LIN {X 0,Y 473.765,Z 475.954,A -85,B 0,C 180,E1 -7294.679,E2 -7294.679} C_VEL
LIN {X 0,Y 473.866,Z 471.994,A -85,B 0,C 180,E1 -7295.958,E2 -7295.958} C_VEL
LIN {X 0,Y 474.033,Z 465.904,A -85,B 0,C 180,E1 -7297.452,E2 -7297.452} C_VEL
LIN {X 0,Y 474.322,Z 459.245,A -85,B 0,C 180,E1 -7298.734,E2 -7298.734} C_VEL
LIN {X 0,Y 474.676,Z 450.981,A -85,B 0,C 180,E1 -7300.017,E2 -7300.017} C_VEL
LIN {X 0,Y 475.049,Z 442.514,A -85,B 0,C 180,E1 -7301.087,E2 -7301.087} C_VEL
LIN {X 0,Y 475.614,Z 432.095,A -85,B 0,C 180,E1 -7302.15,E2 -7302.15} C_VEL
LIN {X 0,Y 476.019,Z 420.854,A -85,B 0,C 180,E1 -7303.075,E2 -7303.075} C_VEL
LIN {X 0,Y 476.498,Z 408.482,A -85,B 0,C 180,E1 -7303.866,E2 -7303.866} C_VEL
LIN {X 0,Y 476.994,Z 396.233,A -85,B 0,C 180,E1 -7304.45,E2 -7304.45} C_VEL
LIN {X 0,Y 477.32,Z 383.727,A -85,B 0,C 180,E1 -7304.876,E2 -7304.876} C_VEL
LIN {X 0,Y 477.558,Z 370.979,A -85,B 0,C 180,E1 -7305.141,E2 -7305.141} C_VEL
LIN {X 0,Y 478.059,Z 286.015,A -85,B 0,C 180,E1 -7306.443,E2 -7306.443} C_VEL
LIN {X 0,Y 475.428,Z 270.249,A -85,B 0,C 180,E1 -7306.808,E2 -7306.808} C_VEL
LIN {X 0,Y 475.47,Z 266.561,A -85,B 0,C 180,E1 -7307.415,E2 -7307.415} C_VEL
LIN {X 0,Y 476.068,Z 250.767,A -85,B 0,C 180,E1 -7310.298,E2 -7310.298} C_VEL
LIN {X 0,Y 476.598,Z 238.624,A -85,B 0,C 180,E1 -7312.543,E2 -7312.543} C_VEL
LIN {X 0,Y 474.683,Z 228.12,A -85,B 0,C 180,E1 -7314.665,E2 -7314.665} C_VEL
LIN {X 0,Y 474.645,Z 227.864,A -85,B 0,C 180,E1 -7315.428,E2 -7315.428} C_VEL
LIN {X 0,Y 474.644,Z 227.861,A -85,B 0,C 180,E1 -7318.281,E2 -7318.281} C_VEL
LIN {X 0,Y 474.6,Z 227.864,A -85,B 0,C 180,E1 -7321.216,E2 -7321.216} C_VEL
LIN {X 0,Y 474.633,Z 227.862,A -85,B 0,C 180,E1 -7324.239,E2 -7324.239} C_VEL
LIN {X 0,Y 474.585,Z 227.866,A -85,B 0,C 180,E1 -7327.382,E2 -7327.382} C_VEL
LIN {X 0,Y 474.615,Z 227.862,A -85,B 0,C 180,E1 -7330.656,E2 -7330.656} C_VEL
LIN {X 0,Y 474.591,Z 227.863,A -85,B 0,C 180,E1 -7333.477,E2 -7333.477} C_VEL
LIN {X 0,Y 474.591,Z 227.861,A -85,B 0,C 180,E1 -7336.518,E2 -7336.518} C_VEL
LIN {X 0,Y 474.593,Z 227.864,A -85,B 0,C 180,E1 -7339.337,E2 -7339.337} C_VEL
LIN {X 0,Y 474.604,Z 227.862,A -85,B 0,C 180,E1 -7341.702,E2 -7341.702} C_VEL
LIN {X 0,Y 474.619,Z 227.867,A -85,B 0,C 180,E1 -7344.723,E2 -7344.723} C_VEL
LIN {X 0,Y 474.631,Z 227.856,A -85,B 0,C 180,E1 -7347.785,E2 -7347.785} C_VEL
LIN {X 0,Y 474.602,Z 227.866,A -85,B 0,C 180,E1 -7350.886,E2 -7350.886} C_VEL
LIN {X 0,Y 474.586,Z 227.863,A -85,B 0,C 180,E1 -7353.621,E2 -7353.621} C_VEL
LIN {X 0,Y 474.628,Z 227.863,A -85,B 0,C 180,E1 -7356.639,E2 -7356.639} C_VEL
LIN {X 0,Y 474.643,Z 227.855,A -85,B 0,C 180,E1 -7360.086,E2 -7360.086} C_VEL
LIN {X 0,Y 474.623,Z 227.863,A -85,B 0,C 180,E1 -7362.771,E2 -7362.771} C_VEL
LIN {X 0,Y 474.623,Z 227.864,A -85,B 0,C 180,E1 -7365.417,E2 -7365.417} C_VEL
LIN {X 0,Y 474.694,Z 227.847,A -85,B 0,C 180,E1 -7368.034,E2 -7368.034} C_VEL
LIN {X 0,Y 474.682,Z 227.853,A -85,B 0,C 180,E1 -7371.483,E2 -7371.483} C_VEL
LIN {X 0,Y 474.743,Z 227.845,A -85,B 0,C 180,E1 -7374.049,E2 -7374.049} C_VEL
LIN {X 0,Y 474.855,Z 227.833,A -85,B 0,C 180,E1 -7377.452,E2 -7377.452} C_VEL
LIN {X 0,Y 474.86,Z 227.83,A -85,B 0,C 180,E1 -7379.997,E2 -7379.997} C_VEL
LIN {X 0,Y 474.856,Z 227.83,A -85,B 0,C 180,E1 -7382.541,E2 -7382.541} C_VEL
LIN {X 0,Y 474.717,Z 227.852,A -85,B 0,C 180,E1 -7385.945,E2 -7385.945} C_VEL
LIN {X 0,Y 474.688,Z 227.85,A -85,B 0,C 180,E1 -7388.511,E2 -7388.511} C_VEL
LIN {X 0,Y 474.683,Z 227.857,A -85,B 0,C 180,E1 -7391.959,E2 -7391.959} C_VEL
LIN {X 0,Y 474.657,Z 227.862,A -85,B 0,C 180,E1 -7395.764,E2 -7395.764} C_VEL
LIN {X 0,Y 474.637,Z 227.857,A -85,B 0,C 180,E1 -7399.007,E2 -7399.007} C_VEL
LIN {X 0,Y 474.562,Z 227.871,A -85,B 0,C 180,E1 -7401.726,E2 -7401.726} C_VEL
LIN {X 0,Y 474.611,Z 227.864,A -85,B 0,C 180,E1 -7404.491,E2 -7404.491} C_VEL
LIN {X 0,Y 474.652,Z 227.856,A -85,B 0,C 180,E1 -7407.331,E2 -7407.331} C_VEL
LIN {X 0,Y 474.573,Z 227.869,A -85,B 0,C 180,E1 -7410.807,E2 -7410.807} C_VEL
LIN {X 0,Y 474.606,Z 227.864,A -85,B 0,C 180,E1 -7413.981,E2 -7413.981} C_VEL
LIN {X 0,Y 474.543,Z 227.875,A -85,B 0,C 180,E1 -7416.897,E2 -7416.897} C_VEL
LIN {X 0,Y 474.62,Z 227.862,A -85,B 0,C 180,E1 -7419.649,E2 -7419.649} C_VEL
LIN {X 0,Y 474.615,Z 227.868,A -85,B 0,C 180,E1 -7422.928,E2 -7422.928} C_VEL
LIN {X 0,Y 474.605,Z 227.868,A -85,B 0,C 180,E1 -7426.243,E2 -7426.243} C_VEL
LIN {X 0,Y 474.634,Z 228.172,A -85,B 0,C 180,E1 -7426.508,E2 -7426.508} C_VEL
LIN {X 0,Y 476.004,Z 235.407,A -85,B 0,C 180,E1 -7428.002,E2 -7428.002} C_VEL
LIN {X 0,Y 475.688,Z 248.758,A -85,B 0,C 180,E1 -7430.56,E2 -7430.56} C_VEL
LIN {X 0,Y 475.414,Z 257.711,A -85,B 0,C 180,E1 -7432.212,E2 -7432.212} C_VEL
LIN {X 0,Y 476.311,Z 262.551,A -85,B 0,C 180,E1 -7432.363,E2 -7432.363} C_VEL
LIN {X 0,Y 478.228,Z 274.047,A -85,B 0,C 180,E1 -7432.616,E2 -7432.616} C_VEL
LIN {X 0,Y 477.488,Z 364.83,A -85,B 0,C 180,E1 -7434.019,E2 -7434.019} C_VEL
LIN {X 0,Y 477.188,Z 378.256,A -85,B 0,C 180,E1 -7434.396,E2 -7434.396} C_VEL
LIN {X 0,Y 476.867,Z 390.684,A -85,B 0,C 180,E1 -7434.918,E2 -7434.918} C_VEL
LIN {X 0,Y 476.416,Z 402.316,A -85,B 0,C 180,E1 -7435.575,E2 -7435.575} C_VEL
LIN {X 0,Y 476.347,Z 403.878,A -85,B 0,C 180,E1 -7435.681,E2 -7435.681} C_VEL
LIN {X 0,Y 475.493,Z 409.056,A -85,B 0,C 180,E1 -7436.025,E2 -7436.025} C_VEL
LIN {X 0,Y 472.367,Z 417.175,A -85,B 0,C 180,E1 -7436.603,E2 -7436.603} C_VEL
LIN {X 0,Y 469.192,Z 424.803,A -85,B 0,C 180,E1 -7437.257,E2 -7437.257} C_VEL
LIN {X 0,Y 468.251,Z 429.193,A -85,B 0,C 180,E1 -7437.72,E2 -7437.72} C_VEL
LIN {X 0,Y 467.764,Z 438.428,A -85,B 0,C 180,E1 -7438.905,E2 -7438.905} C_VEL
LIN {X 0,Y 467.323,Z 446.827,A -85,B 0,C 180,E1 -7440.248,E2 -7440.248} C_VEL
LIN {X 0,Y 467.12,Z 452.975,A -85,B 0,C 180,E1 -7441.467,E2 -7441.467} C_VEL
LIN {X 0,Y 466.95,Z 457.676,A -85,B 0,C 180,E1 -7442.611,E2 -7442.611} C_VEL
LIN {X 0,Y 466.765,Z 462.505,A -85,B 0,C 180,E1 -7444.112,E2 -7444.112} C_VEL
LIN {X 0,Y 466.632,Z 464.816,A -85,B 0,C 180,E1 -7445.059,E2 -7445.059} C_VEL
LIN {X 0,Y 466.503,Z 467.676,A -85,B 0,C 180,E1 -7446.764,E2 -7446.764} C_VEL
LIN {X 0,Y 466.46,Z 468.677,A -85,B 0,C 180,E1 -7447.874,E2 -7447.874} C_VEL
LIN {X 0,Y 466.492,Z 469.047,A -85,B 0,C 180,E1 -7449.063,E2 -7449.063} C_VEL
LIN {X 0,Y 466.512,Z 468.323,A -85,B 0,C 180,E1 -7450.646,E2 -7450.646} C_VEL
LIN {X 0,Y 466.551,Z 467.243,A -85,B 0,C 180,E1 -7451.608,E2 -7451.608} C_VEL
LIN {X 0,Y 466.584,Z 465.864,A -85,B 0,C 180,E1 -7452.469,E2 -7452.469} C_VEL
LIN {X 0,Y 466.737,Z 462.793,A -85,B 0,C 180,E1 -7453.827,E2 -7453.827} C_VEL
LIN {X 0,Y 466.861,Z 458.626,A -85,B 0,C 180,E1 -7455.174,E2 -7455.174} C_VEL
LIN {X 0,Y 467.074,Z 452.208,A -85,B 0,C 180,E1 -7456.736,E2 -7456.736} C_VEL
LIN {X 0,Y 467.434,Z 445.206,A -85,B 0,C 180,E1 -7458.07,E2 -7458.07} C_VEL
LIN {X 0,Y 467.697,Z 438.086,A -85,B 0,C 180,E1 -7459.175,E2 -7459.175} C_VEL
LIN {X 0,Y 468.144,Z 429.45,A -85,B 0,C 180,E1 -7460.278,E2 -7460.278} C_VEL
LIN {X 0,Y 468.644,Z 418.782,A -85,B 0,C 180,E1 -7461.377,E2 -7461.377} C_VEL
LIN {X 0,Y 469.181,Z 408.171,A -85,B 0,C 180,E1 -7462.254,E2 -7462.254} C_VEL
LIN {X 0,Y 469.622,Z 396.505,A -85,B 0,C 180,E1 -7463.017,E2 -7463.017} C_VEL
LIN {X 0,Y 470.048,Z 384.323,A -85,B 0,C 180,E1 -7463.617,E2 -7463.617} C_VEL
LIN {X 0,Y 470.405,Z 371.036,A -85,B 0,C 180,E1 -7464.079,E2 -7464.079} C_VEL
LIN {X 0,Y 470.584,Z 358.189,A -85,B 0,C 180,E1 -7464.35,E2 -7464.35} C_VEL
LIN {X 0,Y 471.037,Z 273.168,A -85,B 0,C 180,E1 -7465.669,E2 -7465.669} C_VEL
LIN {X 0,Y 468.41,Z 258.139,A -85,B 0,C 180,E1 -7466.022,E2 -7466.022} C_VEL
LIN {X 0,Y 468.814,Z 247.613,A -85,B 0,C 180,E1 -7468.068,E2 -7468.068} C_VEL
LIN {X 0,Y 469.142,Z 236.994,A -85,B 0,C 180,E1 -7470.216,E2 -7470.216} C_VEL
LIN {X 0,Y 467.744,Z 228.804,A -85,B 0,C 180,E1 -7472.019,E2 -7472.019} C_VEL
LIN {X 0,Y 467.593,Z 228.742,A -85,B 0,C 180,E1 -7473.448,E2 -7473.448} C_VEL
LIN {X 0,Y 467.696,Z 228.726,A -85,B 0,C 180,E1 -7476.039,E2 -7476.039} C_VEL
LIN {X 0,Y 467.639,Z 228.729,A -85,B 0,C 180,E1 -7478.645,E2 -7478.645} C_VEL
LIN {X 0,Y 467.641,Z 228.73,A -85,B 0,C 180,E1 -7482.147,E2 -7482.147} C_VEL
LIN {X 0,Y 467.609,Z 228.739,A -85,B 0,C 180,E1 -7485.887,E2 -7485.887} C_VEL
LIN {X 0,Y 467.584,Z 228.737,A -85,B 0,C 180,E1 -7489.311,E2 -7489.311} C_VEL
LIN {X 0,Y 467.496,Z 228.753,A -85,B 0,C 180,E1 -7492.077,E2 -7492.077} C_VEL
LIN {X 0,Y 467.533,Z 228.742,A -85,B 0,C 180,E1 -7494.893,E2 -7494.893} C_VEL
LIN {X 0,Y 467.544,Z 228.744,A -85,B 0,C 180,E1 -7497.775,E2 -7497.775} C_VEL
LIN {X 0,Y 467.534,Z 228.742,A -85,B 0,C 180,E1 -7501.048,E2 -7501.048} C_VEL
LIN {X 0,Y 467.544,Z 228.748,A -85,B 0,C 180,E1 -7504.243,E2 -7504.243} C_VEL
LIN {X 0,Y 467.492,Z 228.747,A -85,B 0,C 180,E1 -7507.186,E2 -7507.186} C_VEL
LIN {X 0,Y 467.529,Z 228.747,A -85,B 0,C 180,E1 -7510.271,E2 -7510.271} C_VEL
LIN {X 0,Y 467.521,Z 228.743,A -85,B 0,C 180,E1 -7513.75,E2 -7513.75} C_VEL
LIN {X 0,Y 467.524,Z 228.745,A -85,B 0,C 180,E1 -7516.259,E2 -7516.259} C_VEL
LIN {X 0,Y 467.538,Z 228.741,A -85,B 0,C 180,E1 -7519.738,E2 -7519.738} C_VEL
LIN {X 0,Y 467.529,Z 228.749,A -85,B 0,C 180,E1 -7522.818,E2 -7522.818} C_VEL
LIN {X 0,Y 467.561,Z 228.739,A -85,B 0,C 180,E1 -7525.764,E2 -7525.764} C_VEL
LIN {X 0,Y 467.535,Z 228.748,A -85,B 0,C 180,E1 -7528.964,E2 -7528.964} C_VEL
LIN {X 0,Y 467.534,Z 228.741,A -85,B 0,C 180,E1 -7532.23,E2 -7532.23} C_VEL
LIN {X 0,Y 467.545,Z 228.746,A -85,B 0,C 180,E1 -7535.114,E2 -7535.114} C_VEL
LIN {X 0,Y 467.525,Z 228.745,A -85,B 0,C 180,E1 -7537.93,E2 -7537.93} C_VEL
LIN {X 0,Y 467.615,Z 228.731,A -85,B 0,C 180,E1 -7540.696,E2 -7540.696} C_VEL
LIN {X 0,Y 467.636,Z 228.73,A -85,B 0,C 180,E1 -7544.309,E2 -7544.309} C_VEL
LIN {X 0,Y 467.647,Z 228.735,A -85,B 0,C 180,E1 -7547.858,E2 -7547.858} C_VEL
LIN {X 0,Y 467.638,Z 228.731,A -85,B 0,C 180,E1 -7551.36,E2 -7551.36} C_VEL
LIN {X 0,Y 467.703,Z 228.73,A -85,B 0,C 180,E1 -7553.966,E2 -7553.966} C_VEL
LIN {X 0,Y 467.817,Z 228.707,A -85,B 0,C 180,E1 -7557.42,E2 -7557.42} C_VEL
LIN {X 0,Y 467.854,Z 228.708,A -85,B 0,C 180,E1 -7560.003,E2 -7560.003} C_VEL
LIN {X 0,Y 467.817,Z 228.71,A -85,B 0,C 180,E1 -7562.586,E2 -7562.586} C_VEL
LIN {X 0,Y 467.71,Z 228.724,A -85,B 0,C 180,E1 -7566.041,E2 -7566.041} C_VEL
LIN {X 0,Y 467.644,Z 228.734,A -85,B 0,C 180,E1 -7568.646,E2 -7568.646} C_VEL
LIN {X 0,Y 467.667,Z 228.728,A -85,B 0,C 180,E1 -7572.148,E2 -7572.148} C_VEL
LIN {X 0,Y 467.661,Z 228.726,A -85,B 0,C 180,E1 -7575.887,E2 -7575.887} C_VEL
LIN {X 0,Y 467.633,Z 228.731,A -85,B 0,C 180,E1 -7579.31,E2 -7579.31} C_VEL
LIN {X 0,Y 467.544,Z 228.74,A -85,B 0,C 180,E1 -7582.076,E2 -7582.076} C_VEL
LIN {X 0,Y 467.57,Z 228.745,A -85,B 0,C 180,E1 -7584.892,E2 -7584.892} C_VEL
LIN {X 0,Y 467.56,Z 228.739,A -85,B 0,C 180,E1 -7587.775,E2 -7587.775} C_VEL
LIN {X 0,Y 467.561,Z 228.745,A -85,B 0,C 180,E1 -7591.042,E2 -7591.042} C_VEL
LIN {X 0,Y 467.59,Z 228.734,A -85,B 0,C 180,E1 -7594.241,E2 -7594.241} C_VEL
LIN {X 0,Y 467.556,Z 228.745,A -85,B 0,C 180,E1 -7597.186,E2 -7597.186} C_VEL
LIN {X 0,Y 467.572,Z 228.737,A -85,B 0,C 180,E1 -7600.268,E2 -7600.268} C_VEL
LIN {X 0,Y 467.559,Z 228.745,A -85,B 0,C 180,E1 -7603.746,E2 -7603.746} C_VEL
LIN {X 0,Y 467.558,Z 228.74,A -85,B 0,C 180,E1 -7606.255,E2 -7606.255} C_VEL
LIN {X 0,Y 467.571,Z 228.745,A -85,B 0,C 180,E1 -7609.733,E2 -7609.733} C_VEL
LIN {X 0,Y 467.556,Z 228.739,A -85,B 0,C 180,E1 -7612.815,E2 -7612.815} C_VEL
LIN {X 0,Y 467.598,Z 228.739,A -85,B 0,C 180,E1 -7616.212,E2 -7616.212} C_VEL
LIN {X 0,Y 467.58,Z 228.736,A -85,B 0,C 180,E1 -7619.266,E2 -7619.266} C_VEL
LIN {X 0,Y 467.617,Z 228.738,A -85,B 0,C 180,E1 -7622.468,E2 -7622.468} C_VEL
LIN {X 0,Y 467.639,Z 228.933,A -85,B 0,C 180,E1 -7625.202,E2 -7625.202} C_VEL
LIN {X 0,Y 469.538,Z 239.426,A -85,B 0,C 180,E1 -7627.329,E2 -7627.329} C_VEL
LIN {X 0,Y 469.006,Z 254.014,A -85,B 0,C 180,E1 -7630.067,E2 -7630.067} C_VEL
LIN {X 0,Y 468.383,Z 270.156,A -85,B 0,C 180,E1 -7633.013,E2 -7633.013} C_VEL
LIN {X 0,Y 471.181,Z 288.676,A -85,B 0,C 180,E1 -7633.429,E2 -7633.429} C_VEL
LIN {X 0,Y 470.481,Z 377.791,A -85,B 0,C 180,E1 -7634.817,E2 -7634.817} C_VEL
LIN {X 0,Y 470.119,Z 391.064,A -85,B 0,C 180,E1 -7635.193,E2 -7635.193} C_VEL
LIN {X 0,Y 469.669,Z 404.363,A -85,B 0,C 180,E1 -7635.76,E2 -7635.76} C_VEL
LIN {X 0,Y 469.2,Z 416.796,A -85,B 0,C 180,E1 -7636.497,E2 -7636.497} C_VEL
LIN {X 0,Y 468.768,Z 427.881,A -85,B 0,C 180,E1 -7637.341,E2 -7637.341} C_VEL
LIN {X 0,Y 468.257,Z 438.115,A -85,B 0,C 180,E1 -7638.309,E2 -7638.309} C_VEL
LIN {X 0,Y 467.772,Z 447.372,A -85,B 0,C 180,E1 -7639.393,E2 -7639.393} C_VEL
LIN {X 0,Y 467.341,Z 456.36,A -85,B 0,C 180,E1 -7640.695,E2 -7640.695} C_VEL
LIN {X 0,Y 467.057,Z 463.597,A -85,B 0,C 180,E1 -7641.998,E2 -7641.998} C_VEL
LIN {X 0,Y 466.862,Z 468.48,A -85,B 0,C 180,E1 -7643.082,E2 -7643.082} C_VEL
LIN {X 0,Y 466.793,Z 473.226,A -85,B 0,C 180,E1 -7644.383,E2 -7644.383} C_VEL
LIN {X 0,Y 466.65,Z 476.851,A -85,B 0,C 180,E1 -7645.68,E2 -7645.68} C_VEL
LIN {X 0,Y 466.663,Z 478.725,A -85,B 0,C 180,E1 -7646.545,E2 -7646.545} C_VEL
LIN {X 0,Y 466.647,Z 480.132,A -85,B 0,C 180,E1 -7647.409,E2 -7647.409} C_VEL
LIN {X 0,Y 466.592,Z 481.747,A -85,B 0,C 180,E1 -7649.136,E2 -7649.136} C_VEL
LIN {X 0,Y 466.601,Z 481.972,A -85,B 0,C 180,E1 -7649.999,E2 -7649.999} C_VEL
LIN {X 0,Y 466.592,Z 481.766,A -85,B 0,C 180,E1 -7650.862,E2 -7650.862} C_VEL
LIN {X 0,Y 466.646,Z 480.176,A -85,B 0,C 180,E1 -7652.588,E2 -7652.588} C_VEL
LIN {X 0,Y 466.663,Z 478.789,A -85,B 0,C 180,E1 -7653.452,E2 -7653.452} C_VEL
LIN {X 0,Y 466.693,Z 475.866,A -85,B 0,C 180,E1 -7654.75,E2 -7654.75} C_VEL
LIN {X 0,Y 466.78,Z 471.908,A -85,B 0,C 180,E1 -7656.048,E2 -7656.048} C_VEL
LIN {X 0,Y 466.983,Z 465.823,A -85,B 0,C 180,E1 -7657.566,E2 -7657.566} C_VEL
LIN {X 0,Y 467.288,Z 459.175,A -85,B 0,C 180,E1 -7658.867,E2 -7658.867} C_VEL
LIN {X 0,Y 467.636,Z 450.933,A -85,B 0,C 180,E1 -7660.17,E2 -7660.17} C_VEL
LIN {X 0,Y 468.084,Z 442.497,A -85,B 0,C 180,E1 -7661.254,E2 -7661.254} C_VEL
LIN {X 0,Y 468.658,Z 432.316,A -85,B 0,C 180,E1 -7662.315,E2 -7662.315} C_VEL
LIN {X 0,Y 469.022,Z 422.073,A -85,B 0,C 180,E1 -7663.186,E2 -7663.186} C_VEL
LIN {X 0,Y 469.529,Z 410.519,A -85,B 0,C 180,E1 -7663.965,E2 -7663.965} C_VEL
LIN {X 0,Y 470.047,Z 399.055,A -85,B 0,C 180,E1 -7664.557,E2 -7664.557} C_VEL
LIN {X 0,Y 470.387,Z 385.936,A -85,B 0,C 180,E1 -7665.045,E2 -7665.045} C_VEL
LIN {X 0,Y 470.747,Z 373.321,A -85,B 0,C 180,E1 -7665.338,E2 -7665.338} C_VEL
LIN {X 0,Y 471.274,Z 286.938,A -85,B 0,C 180,E1 -7666.686,E2 -7666.686} C_VEL
LIN {X 0,Y 468.441,Z 269.969,A -85,B 0,C 180,E1 -7667.094,E2 -7667.094} C_VEL
LIN {X 0,Y 469.038,Z 254.391,A -85,B 0,C 180,E1 -7669.929,E2 -7669.929} C_VEL
LIN {X 0,Y 469.657,Z 239.86,A -85,B 0,C 180,E1 -7672.662,E2 -7672.662} C_VEL
LIN {X 0,Y 467.677,Z 229.048,A -85,B 0,C 180,E1 -7674.881,E2 -7674.881} C_VEL
LIN {X 0,Y 467.616,Z 228.739,A -85,B 0,C 180,E1 -7675.306,E2 -7675.306} C_VEL
LIN {X 0,Y 467.619,Z 228.739,A -85,B 0,C 180,E1 -7677.767,E2 -7677.767} C_VEL
LIN {X 0,Y 467.569,Z 228.739,A -85,B 0,C 180,E1 -7681.042,E2 -7681.042} C_VEL
LIN {X 0,Y 467.59,Z 228.739,A -85,B 0,C 180,E1 -7684.24,E2 -7684.24} C_VEL
LIN {X 0,Y 467.543,Z 228.743,A -85,B 0,C 180,E1 -7687.183,E2 -7687.183} C_VEL
LIN {X 0,Y 467.57,Z 228.744,A -85,B 0,C 180,E1 -7690.263,E2 -7690.263} C_VEL
LIN {X 0,Y 467.561,Z 228.741,A -85,B 0,C 180,E1 -7692.561,E2 -7692.561} C_VEL
LIN {X 0,Y 467.565,Z 228.738,A -85,B 0,C 180,E1 -7695.05,E2 -7695.05} C_VEL
LIN {X 0,Y 467.565,Z 228.745,A -85,B 0,C 180,E1 -7698.593,E2 -7698.593} C_VEL
LIN {X 0,Y 467.559,Z 228.741,A -85,B 0,C 180,E1 -7701.952,E2 -7701.952} C_VEL
LIN {X 0,Y 467.559,Z 228.741,A -85,B 0,C 180,E1 -7705.164,E2 -7705.164} C_VEL
LIN {X 0,Y 467.578,Z 228.738,A -85,B 0,C 180,E1 -7708.257,E2 -7708.257} C_VEL
LIN {X 0,Y 467.549,Z 228.742,A -85,B 0,C 180,E1 -7711.246,E2 -7711.246} C_VEL
LIN {X 0,Y 467.562,Z 228.739,A -85,B 0,C 180,E1 -7714.155,E2 -7714.155} C_VEL
LIN {X 0,Y 467.565,Z 228.745,A -85,B 0,C 180,E1 -7716.993,E2 -7716.993} C_VEL
LIN {X 0,Y 467.613,Z 228.731,A -85,B 0,C 180,E1 -7719.774,E2 -7719.774} C_VEL
LIN {X 0,Y 467.585,Z 228.737,A -85,B 0,C 180,E1 -7722.503,E2 -7722.503} C_VEL
LIN {X 0,Y 467.585,Z 228.744,A -85,B 0,C 180,E1 -7725.193,E2 -7725.193} C_VEL
LIN {X 0,Y 467.646,Z 228.726,A -85,B 0,C 180,E1 -7727.851,E2 -7727.851} C_VEL
LIN {X 0,Y 467.642,Z 228.732,A -85,B 0,C 180,E1 -7731.353,E2 -7731.353} C_VEL
LIN {X 0,Y 467.708,Z 228.722,A -85,B 0,C 180,E1 -7733.959,E2 -7733.959} C_VEL
LIN {X 0,Y 467.795,Z 228.712,A -85,B 0,C 180,E1 -7737.414,E2 -7737.414} C_VEL
LIN {X 0,Y 467.83,Z 228.706,A -85,B 0,C 180,E1 -7739.997,E2 -7739.997} C_VEL
LIN {X 0,Y 467.797,Z 228.709,A -85,B 0,C 180,E1 -7742.58,E2 -7742.58} C_VEL
LIN {X 0,Y 467.682,Z 228.727,A -85,B 0,C 180,E1 -7746.035,E2 -7746.035} C_VEL
LIN {X 0,Y 467.647,Z 228.727,A -85,B 0,C 180,E1 -7748.64,E2 -7748.64} C_VEL
LIN {X 0,Y 467.635,Z 228.732,A -85,B 0,C 180,E1 -7752.142,E2 -7752.142} C_VEL
LIN {X 0,Y 467.626,Z 228.737,A -85,B 0,C 180,E1 -7755.881,E2 -7755.881} C_VEL
LIN {X 0,Y 467.596,Z 228.735,A -85,B 0,C 180,E1 -7759.305,E2 -7759.305} C_VEL
LIN {X 0,Y 467.508,Z 228.752,A -85,B 0,C 180,E1 -7762.071,E2 -7762.071} C_VEL
LIN {X 0,Y 467.556,Z 228.739,A -85,B 0,C 180,E1 -7764.885,E2 -7764.885} C_VEL
LIN {X 0,Y 467.591,Z 228.737,A -85,B 0,C 180,E1 -7767.766,E2 -7767.766} C_VEL
LIN {X 0,Y 467.537,Z 228.744,A -85,B 0,C 180,E1 -7771.042,E2 -7771.042} C_VEL
LIN {X 0,Y 467.558,Z 228.745,A -85,B 0,C 180,E1 -7774.24,E2 -7774.24} C_VEL
LIN {X 0,Y 467.518,Z 228.747,A -85,B 0,C 180,E1 -7777.184,E2 -7777.184} C_VEL
LIN {X 0,Y 467.562,Z 228.744,A -85,B 0,C 180,E1 -7780.26,E2 -7780.26} C_VEL
LIN {X 0,Y 467.583,Z 228.742,A -85,B 0,C 180,E1 -7782.569,E2 -7782.569} C_VEL
LIN {X 0,Y 467.589,Z 228.823,A -85,B 0,C 180,E1 -7786.214,E2 -7786.214} C_VEL
LIN {X 0,Y 469.088,Z 236.967,A -85,B 0,C 180,E1 -7787.953,E2 -7787.953} C_VEL
LIN {X 0,Y 468.743,Z 249.657,A -85,B 0,C 180,E1 -7790.418,E2 -7790.418} C_VEL
LIN {X 0,Y 468.48,Z 257.715,A -85,B 0,C 180,E1 -7791.928,E2 -7791.928} C_VEL
LIN {X 0,Y 468.99,Z 260.702,A -85,B 0,C 180,E1 -7792.045,E2 -7792.045} C_VEL
LIN {X 0,Y 471.426,Z 273.939,A -85,B 0,C 180,E1 -7792.353,E2 -7792.353} C_VEL
LIN {X 0,Y 470.659,Z 365.908,A -85,B 0,C 180,E1 -7793.804,E2 -7793.804} C_VEL
LIN {X 0,Y 470.329,Z 379.436,A -85,B 0,C 180,E1 -7794.202,E2 -7794.202} C_VEL
LIN {X 0,Y 470.01,Z 391.404,A -85,B 0,C 180,E1 -7794.723,E2 -7794.723} C_VEL
LIN {X 0,Y 469.507,Z 403.103,A -85,B 0,C 180,E1 -7795.406,E2 -7795.406} C_VEL
LIN {X 0,Y 468.978,Z 413.717,A -85,B 0,C 180,E1 -7796.198,E2 -7796.198} C_VEL
LIN {X 0,Y 468.514,Z 423.803,A -85,B 0,C 180,E1 -7797.134,E2 -7797.134} C_VEL
LIN {X 0,Y 468.251,Z 429.193,A -85,B 0,C 180,E1 -7797.72,E2 -7797.72} C_VEL
LIN {X 0,Y 467.306,Z 433.457,A -85,B 0,C 180,E1 -7798.21,E2 -7798.21} C_VEL
LIN {X 0,Y 464.097,Z 440.035,A -85,B 0,C 180,E1 -7799.037,E2 -7799.037} C_VEL
LIN {X 0,Y 461.001,Z 445.992,A -85,B 0,C 180,E1 -7799.94,E2 -7799.94} C_VEL
LIN {X 0,Y 460.238,Z 449.28,A -85,B 0,C 180,E1 -7800.542,E2 -7800.542} C_VEL
LIN {X 0,Y 460.004,Z 454.792,A -85,B 0,C 180,E1 -7801.732,E2 -7801.732} C_VEL
LIN {X 0,Y 459.78,Z 460.175,A -85,B 0,C 180,E1 -7803.199,E2 -7803.199} C_VEL
LIN {X 0,Y 459.599,Z 464.172,A -85,B 0,C 180,E1 -7804.651,E2 -7804.651} C_VEL
LIN {X 0,Y 459.486,Z 466.143,A -85,B 0,C 180,E1 -7805.61,E2 -7805.61} C_VEL
LIN {X 0,Y 459.428,Z 467.622,A -85,B 0,C 180,E1 -7806.598,E2 -7806.598} C_VEL
LIN {X 0,Y 459.37,Z 468.565,A -85,B 0,C 180,E1 -7807.514,E2 -7807.514} C_VEL
LIN {X 0,Y 459.404,Z 469.136,A -85,B 0,C 180,E1 -7808.921,E2 -7808.921} C_VEL
LIN {X 0,Y 459.43,Z 468.684,A -85,B 0,C 180,E1 -7810.336,E2 -7810.336} C_VEL
LIN {X 0,Y 459.45,Z 467.524,A -85,B 0,C 180,E1 -7811.494,E2 -7811.494} C_VEL
LIN {X 0,Y 459.541,Z 464.751,A -85,B 0,C 180,E1 -7813.109,E2 -7813.109} C_VEL
LIN {X 0,Y 459.696,Z 461.507,A -85,B 0,C 180,E1 -7814.38,E2 -7814.38} C_VEL
LIN {X 0,Y 459.849,Z 456.545,A -85,B 0,C 180,E1 -7815.847,E2 -7815.847} C_VEL
LIN {X 0,Y 460.167,Z 449.428,A -85,B 0,C 180,E1 -7817.431,E2 -7817.431} C_VEL
LIN {X 0,Y 460.513,Z 441.734,A -85,B 0,C 180,E1 -7818.781,E2 -7818.781} C_VEL
LIN {X 0,Y 460.934,Z 433.851,A -85,B 0,C 180,E1 -7819.903,E2 -7819.903} C_VEL
LIN {X 0,Y 461.399,Z 424.226,A -85,B 0,C 180,E1 -7821.019,E2 -7821.019} C_VEL
LIN {X 0,Y 461.953,Z 413.581,A -85,B 0,C 180,E1 -7822.016,E2 -7822.016} C_VEL
LIN {X 0,Y 462.457,Z 403.178,A -85,B 0,C 180,E1 -7822.799,E2 -7822.799} C_VEL
LIN {X 0,Y 462.968,Z 390.897,A -85,B 0,C 180,E1 -7823.519,E2 -7823.519} C_VEL
LIN {X 0,Y 463.308,Z 378.046,A -85,B 0,C 180,E1 -7824.07,E2 -7824.07} C_VEL
LIN {X 0,Y 463.638,Z 365.538,A -85,B 0,C 180,E1 -7824.429,E2 -7824.429} C_VEL
LIN {X 0,Y 464.212,Z 273.918,A -85,B 0,C 180,E1 -7825.891,E2 -7825.891} C_VEL
LIN {X 0,Y 461.43,Z 258.269,A -85,B 0,C 180,E1 -7826.263,E2 -7826.263} C_VEL
LIN {X 0,Y 461.672,Z 252.419,A -85,B 0,C 180,E1 -7827.384,E2 -7827.384} C_VEL
LIN {X 0,Y 462.213,Z 239.599,A -85,B 0,C 180,E1 -7830.001,E2 -7830.001} C_VEL
LIN {X 0,Y 461.573,Z 234.503,A -85,B 0,C 180,E1 -7831.092,E2 -7831.092} C_VEL
LIN {X 0,Y 460.711,Z 229.692,A -85,B 0,C 180,E1 -7832.187,E2 -7832.187} C_VEL
LIN {X 0,Y 460.654,Z 229.607,A -85,B 0,C 180,E1 -7835.253,E2 -7835.253} C_VEL
LIN {X 0,Y 460.653,Z 229.602,A -85,B 0,C 180,E1 -7837.893,E2 -7837.893} C_VEL
LIN {X 0,Y 460.587,Z 229.613,A -85,B 0,C 180,E1 -7841.443,E2 -7841.443} C_VEL
LIN {X 0,Y 460.511,Z 229.619,A -85,B 0,C 180,E1 -7844.135,E2 -7844.135} C_VEL
LIN {X 0,Y 460.524,Z 229.615,A -85,B 0,C 180,E1 -7846.857,E2 -7846.857} C_VEL
LIN {X 0,Y 460.53,Z 229.619,A -85,B 0,C 180,E1 -7849.618,E2 -7849.618} C_VEL
LIN {X 0,Y 460.473,Z 229.624,A -85,B 0,C 180,E1 -7852.432,E2 -7852.432} C_VEL
LIN {X 0,Y 460.51,Z 229.621,A -85,B 0,C 180,E1 -7855.799,E2 -7855.799} C_VEL
LIN {X 0,Y 460.491,Z 229.626,A -85,B 0,C 180,E1 -7858.238,E2 -7858.238} C_VEL
LIN {X 0,Y 460.488,Z 229.619,A -85,B 0,C 180,E1 -7861.286,E2 -7861.286} C_VEL
LIN {X 0,Y 460.489,Z 229.626,A -85,B 0,C 180,E1 -7864.507,E2 -7864.507} C_VEL
LIN {X 0,Y 460.456,Z 229.623,A -85,B 0,C 180,E1 -7867.629,E2 -7867.629} C_VEL
LIN {X 0,Y 460.489,Z 229.622,A -85,B 0,C 180,E1 -7871.017,E2 -7871.017} C_VEL
LIN {X 0,Y 460.487,Z 229.627,A -85,B 0,C 180,E1 -7874.594,E2 -7874.594} C_VEL
LIN {X 0,Y 460.47,Z 229.621,A -85,B 0,C 180,E1 -7877.819,E2 -7877.819} C_VEL
LIN {X 0,Y 460.493,Z 229.619,A -85,B 0,C 180,E1 -7880.14,E2 -7880.14} C_VEL
LIN {X 0,Y 460.459,Z 229.625,A -85,B 0,C 180,E1 -7883.475,E2 -7883.475} C_VEL
LIN {X 0,Y 460.501,Z 229.621,A -85,B 0,C 180,E1 -7886.678,E2 -7886.678} C_VEL
LIN {X 0,Y 460.49,Z 229.62,A -85,B 0,C 180,E1 -7889.764,E2 -7889.764} C_VEL
LIN {X 0,Y 460.478,Z 229.623,A -85,B 0,C 180,E1 -7892.755,E2 -7892.755} C_VEL
LIN {X 0,Y 460.507,Z 229.621,A -85,B 0,C 180,E1 -7895.671,E2 -7895.671} C_VEL
LIN {X 0,Y 460.516,Z 229.616,A -85,B 0,C 180,E1 -7898.583,E2 -7898.583} C_VEL
LIN {X 0,Y 460.579,Z 229.613,A -85,B 0,C 180,E1 -7901.315,E2 -7901.315} C_VEL
LIN {X 0,Y 460.584,Z 229.61,A -85,B 0,C 180,E1 -7904.062,E2 -7904.062} C_VEL
LIN {X 0,Y 460.603,Z 229.613,A -85,B 0,C 180,E1 -7907.67,E2 -7907.67} C_VEL
LIN {X 0,Y 460.593,Z 229.607,A -85,B 0,C 180,E1 -7911.227,E2 -7911.227} C_VEL
LIN {X 0,Y 460.67,Z 229.604,A -85,B 0,C 180,E1 -7913.873,E2 -7913.873} C_VEL
LIN {X 0,Y 460.761,Z 229.586,A -85,B 0,C 180,E1 -7917.381,E2 -7917.381} C_VEL
LIN {X 0,Y 460.824,Z 229.584,A -85,B 0,C 180,E1 -7920.003,E2 -7920.003} C_VEL
LIN {X 0,Y 460.761,Z 229.589,A -85,B 0,C 180,E1 -7922.626,E2 -7922.626} C_VEL
LIN {X 0,Y 460.676,Z 229.601,A -85,B 0,C 180,E1 -7926.134,E2 -7926.134} C_VEL
LIN {X 0,Y 460.599,Z 229.609,A -85,B 0,C 180,E1 -7928.78,E2 -7928.78} C_VEL
LIN {X 0,Y 460.621,Z 229.608,A -85,B 0,C 180,E1 -7932.337,E2 -7932.337} C_VEL
LIN {X 0,Y 460.614,Z 229.604,A -85,B 0,C 180,E1 -7936,E2 -7936} C_VEL
LIN {X 0,Y 460.579,Z 229.608,A -85,B 0,C 180,E1 -7939.618,E2 -7939.618} C_VEL
LIN {X 0,Y 460.521,Z 229.618,A -85,B 0,C 180,E1 -7942.431,E2 -7942.431} C_VEL
LIN {X 0,Y 460.547,Z 229.612,A -85,B 0,C 180,E1 -7945.794,E2 -7945.794} C_VEL
LIN {X 0,Y 460.534,Z 229.621,A -85,B 0,C 180,E1 -7949.234,E2 -7949.234} C_VEL
LIN {X 0,Y 460.532,Z 229.614,A -85,B 0,C 180,E1 -7952.287,E2 -7952.287} C_VEL
LIN {X 0,Y 460.519,Z 229.622,A -85,B 0,C 180,E1 -7955.447,E2 -7955.447} C_VEL
LIN {X 0,Y 460.518,Z 229.617,A -85,B 0,C 180,E1 -7958.892,E2 -7958.892} C_VEL
LIN {X 0,Y 460.517,Z 229.623,A -85,B 0,C 180,E1 -7961.599,E2 -7961.599} C_VEL
LIN {X 0,Y 460.525,Z 229.614,A -85,B 0,C 180,E1 -7964.59,E2 -7964.59} C_VEL
LIN {X 0,Y 460.489,Z 229.627,A -85,B 0,C 180,E1 -7967.813,E2 -7967.813} C_VEL
LIN {X 0,Y 460.526,Z 229.618,A -85,B 0,C 180,E1 -7970.136,E2 -7970.136} C_VEL
LIN {X 0,Y 460.486,Z 229.622,A -85,B 0,C 180,E1 -7973.47,E2 -7973.47} C_VEL
LIN {X 0,Y 460.542,Z 229.613,A -85,B 0,C 180,E1 -7976.675,E2 -7976.675} C_VEL
LIN {X 0,Y 460.52,Z 229.619,A -85,B 0,C 180,E1 -7979.759,E2 -7979.759} C_VEL
LIN {X 0,Y 460.547,Z 229.619,A -85,B 0,C 180,E1 -7982.753,E2 -7982.753} C_VEL
LIN {X 0,Y 460.594,Z 229.796,A -85,B 0,C 180,E1 -7985.008,E2 -7985.008} C_VEL
LIN {X 0,Y 462.556,Z 240.445,A -85,B 0,C 180,E1 -7987.203,E2 -7987.203} C_VEL
LIN {X 0,Y 462.146,Z 251.389,A -85,B 0,C 180,E1 -7989.293,E2 -7989.293} C_VEL
LIN {X 0,Y 461.521,Z 265.951,A -85,B 0,C 180,E1 -7992.038,E2 -7992.038} C_VEL
LIN {X 0,Y 461.396,Z 270.235,A -85,B 0,C 180,E1 -7992.776,E2 -7992.776} C_VEL
LIN {X 0,Y 464.359,Z 288.708,A -85,B 0,C 180,E1 -7993.191,E2 -7993.191} C_VEL
LIN {X 0,Y 463.583,Z 378.085,A -85,B 0,C 180,E1 -7994.614,E2 -7994.614} C_VEL
LIN {X 0,Y 463.187,Z 391.99,A -85,B 0,C 180,E1 -7995.023,E2 -7995.023} C_VEL
LIN {X 0,Y 462.73,Z 404.96,A -85,B 0,C 180,E1 -7995.598,E2 -7995.598} C_VEL
LIN {X 0,Y 462.226,Z 417.548,A -85,B 0,C 180,E1 -7996.367,E2 -7996.367} C_VEL
LIN {X 0,Y 461.782,Z 428.246,A -85,B 0,C 180,E1 -7997.204,E2 -7997.204} C_VEL
LIN {X 0,Y 461.26,Z 437.844,A -85,B 0,C 180,E1 -7998.129,E2 -7998.129} C_VEL
LIN {X 0,Y 460.773,Z 447.148,A -85,B 0,C 180,E1 -7999.23,E2 -7999.23} C_VEL
LIN {X 0,Y 460.297,Z 456.169,A -85,B 0,C 180,E1 -8000.552,E2 -8000.552} C_VEL
LIN {X 0,Y 460.013,Z 463.433,A -85,B 0,C 180,E1 -8001.874,E2 -8001.874} C_VEL
LIN {X 0,Y 459.782,Z 468.333,A -85,B 0,C 180,E1 -8002.975,E2 -8002.975} C_VEL
LIN {X 0,Y 459.691,Z 473.094,A -85,B 0,C 180,E1 -8004.295,E2 -8004.295} C_VEL
LIN {X 0,Y 459.568,Z 476.731,A -85,B 0,C 180,E1 -8005.613,E2 -8005.613} C_VEL
LIN {X 0,Y 459.56,Z 478.61,A -85,B 0,C 180,E1 -8006.492,E2 -8006.492} C_VEL
LIN {X 0,Y 459.569,Z 480.024,A -85,B 0,C 180,E1 -8007.369,E2 -8007.369} C_VEL
LIN {X 0,Y 459.497,Z 481.644,A -85,B 0,C 180,E1 -8009.122,E2 -8009.122} C_VEL
LIN {X 0,Y 459.504,Z 481.873,A -85,B 0,C 180,E1 -8009.999,E2 -8009.999} C_VEL
LIN {X 0,Y 459.497,Z 481.671,A -85,B 0,C 180,E1 -8010.875,E2 -8010.875} C_VEL
LIN {X 0,Y 459.569,Z 480.088,A -85,B 0,C 180,E1 -8012.628,E2 -8012.628} C_VEL
LIN {X 0,Y 459.56,Z 478.706,A -85,B 0,C 180,E1 -8013.506,E2 -8013.506} C_VEL
LIN {X 0,Y 459.625,Z 475.792,A -85,B 0,C 180,E1 -8014.823,E2 -8014.823} C_VEL
LIN {X 0,Y 459.704,Z 471.848,A -85,B 0,C 180,E1 -8016.142,E2 -8016.142} C_VEL
LIN {X 0,Y 459.871,Z 466.774,A -85,B 0,C 180,E1 -8017.462,E2 -8017.462} C_VEL
LIN {X 0,Y 460.175,Z 460.392,A -85,B 0,C 180,E1 -8018.783,E2 -8018.783} C_VEL
LIN {X 0,Y 460.572,Z 452.42,A -85,B 0,C 180,E1 -8020.105,E2 -8020.105} C_VEL
LIN {X 0,Y 460.97,Z 444.305,A -85,B 0,C 180,E1 -8021.207,E2 -8021.207} C_VEL
LIN {X 0,Y 461.558,Z 434.413,A -85,B 0,C 180,E1 -8022.307,E2 -8022.307} C_VEL
LIN {X 0,Y 462.063,Z 423.443,A -85,B 0,C 180,E1 -8023.287,E2 -8023.287} C_VEL
LIN {X 0,Y 462.583,Z 412.416,A -85,B 0,C 180,E1 -8024.067,E2 -8024.067} C_VEL
LIN {X 0,Y 463.156,Z 400.404,A -85,B 0,C 180,E1 -8024.723,E2 -8024.723} C_VEL
LIN {X 0,Y 463.509,Z 388.122,A -85,B 0,C 180,E1 -8025.217,E2 -8025.217} C_VEL
LIN {X 0,Y 463.907,Z 375.514,A -85,B 0,C 180,E1 -8025.541,E2 -8025.541} C_VEL
LIN {X 0,Y 464.481,Z 287.566,A -85,B 0,C 180,E1 -8026.943,E2 -8026.943} C_VEL
LIN {X 0,Y 461.496,Z 269.83,A -85,B 0,C 180,E1 -8027.38,E2 -8027.38} C_VEL
LIN {X 0,Y 462.131,Z 254.416,A -85,B 0,C 180,E1 -8030.24,E2 -8030.24} C_VEL
LIN {X 0,Y 462.747,Z 242.307,A -85,B 0,C 180,E1 -8032.548,E2 -8032.548} C_VEL
LIN {X 0,Y 461.654,Z 235.11,A -85,B 0,C 180,E1 -8034.016,E2 -8034.016} C_VEL
LIN {X 0,Y 460.6,Z 229.778,A -85,B 0,C 180,E1 -8035.17,E2 -8035.17} C_VEL
LIN {X 0,Y 460.552,Z 229.617,A -85,B 0,C 180,E1 -8038.231,E2 -8038.231} C_VEL
LIN {X 0,Y 460.523,Z 229.619,A -85,B 0,C 180,E1 -8041.28,E2 -8041.28} C_VEL
LIN {X 0,Y 460.533,Z 229.615,A -85,B 0,C 180,E1 -8044.503,E2 -8044.503} C_VEL
LIN {X 0,Y 460.499,Z 229.623,A -85,B 0,C 180,E1 -8047.621,E2 -8047.621} C_VEL
LIN {X 0,Y 460.528,Z 229.614,A -85,B 0,C 180,E1 -8051.009,E2 -8051.009} C_VEL
LIN {X 0,Y 460.512,Z 229.621,A -85,B 0,C 180,E1 -8054.587,E2 -8054.587} C_VEL
LIN {X 0,Y 460.501,Z 229.615,A -85,B 0,C 180,E1 -8057.814,E2 -8057.814} C_VEL
LIN {X 0,Y 460.512,Z 229.623,A -85,B 0,C 180,E1 -8060.133,E2 -8060.133} C_VEL
LIN {X 0,Y 460.47,Z 229.621,A -85,B 0,C 180,E1 -8063.467,E2 -8063.467} C_VEL
LIN {X 0,Y 460.524,Z 229.619,A -85,B 0,C 180,E1 -8066.672,E2 -8066.672} C_VEL
LIN {X 0,Y 460.502,Z 229.618,A -85,B 0,C 180,E1 -8069.757,E2 -8069.757} C_VEL
LIN {X 0,Y 460.525,Z 229.624,A -85,B 0,C 180,E1 -8072.75,E2 -8072.75} C_VEL
LIN {X 0,Y 460.512,Z 229.617,A -85,B 0,C 180,E1 -8075.663,E2 -8075.663} C_VEL
LIN {X 0,Y 460.515,Z 229.62,A -85,B 0,C 180,E1 -8078.575,E2 -8078.575} C_VEL
LIN {X 0,Y 460.577,Z 229.613,A -85,B 0,C 180,E1 -8081.308,E2 -8081.308} C_VEL
LIN {X 0,Y 460.597,Z 229.604,A -85,B 0,C 180,E1 -8084.056,E2 -8084.056} C_VEL
LIN {X 0,Y 460.599,Z 229.605,A -85,B 0,C 180,E1 -8087.663,E2 -8087.663} C_VEL
LIN {X 0,Y 460.592,Z 229.612,A -85,B 0,C 180,E1 -8091.22,E2 -8091.22} C_VEL
LIN {X 0,Y 460.674,Z 229.599,A -85,B 0,C 180,E1 -8093.866,E2 -8093.866} C_VEL
LIN {X 0,Y 460.739,Z 229.59,A -85,B 0,C 180,E1 -8097.374,E2 -8097.374} C_VEL
LIN {X 0,Y 460.779,Z 229.584,A -85,B 0,C 180,E1 -8099.997,E2 -8099.997} C_VEL
LIN {X 0,Y 460.741,Z 229.588,A -85,B 0,C 180,E1 -8102.619,E2 -8102.619} C_VEL
LIN {X 0,Y 460.648,Z 229.602,A -85,B 0,C 180,E1 -8106.127,E2 -8106.127} C_VEL
LIN {X 0,Y 460.597,Z 229.605,A -85,B 0,C 180,E1 -8108.773,E2 -8108.773} C_VEL
LIN {X 0,Y 460.576,Z 229.609,A -85,B 0,C 180,E1 -8112.432,E2 -8112.432} C_VEL
LIN {X 0,Y 460.578,Z 229.614,A -85,B 0,C 180,E1 -8115.994,E2 -8115.994} C_VEL
LIN {X 0,Y 460.542,Z 229.616,A -85,B 0,C 180,E1 -8119.612,E2 -8119.612} C_VEL
LIN {X 0,Y 460.484,Z 229.624,A -85,B 0,C 180,E1 -8122.425,E2 -8122.425} C_VEL
LIN {X 0,Y 460.524,Z 229.617,A -85,B 0,C 180,E1 -8125.795,E2 -8125.795} C_VEL
LIN {X 0,Y 460.523,Z 229.616,A -85,B 0,C 180,E1 -8128.23,E2 -8128.23} C_VEL
LIN {X 0,Y 460.489,Z 229.621,A -85,B 0,C 180,E1 -8131.28,E2 -8131.28} C_VEL
LIN {X 0,Y 460.502,Z 229.625,A -85,B 0,C 180,E1 -8134.503,E2 -8134.503} C_VEL
LIN {X 0,Y 460.497,Z 229.621,A -85,B 0,C 180,E1 -8137.618,E2 -8137.618} C_VEL
LIN {X 0,Y 460.525,Z 229.621,A -85,B 0,C 180,E1 -8140.27,E2 -8140.27} C_VEL
LIN {X 0,Y 460.488,Z 229.624,A -85,B 0,C 180,E1 -8143.37,E2 -8143.37} C_VEL
LIN {X 0,Y 460.519,Z 229.696,A -85,B 0,C 180,E1 -8145.979,E2 -8145.979} C_VEL
LIN {X 0,Y 462.079,Z 237.738,A -85,B 0,C 180,E1 -8147.74,E2 -8147.74} C_VEL
LIN {X 0,Y 461.972,Z 244.832,A -85,B 0,C 180,E1 -8149.146,E2 -8149.146} C_VEL
LIN {X 0,Y 461.57,Z 257.948,A -85,B 0,C 180,E1 -8151.663,E2 -8151.663} C_VEL
LIN {X 0,Y 463.248,Z 266.658,A -85,B 0,C 180,E1 -8151.908,E2 -8151.908} C_VEL
LIN {X 0,Y 464.659,Z 274.599,A -85,B 0,C 180,E1 -8152.095,E2 -8152.095} C_VEL
LIN {X 0,Y 463.857,Z 365.807,A -85,B 0,C 180,E1 -8153.555,E2 -8153.555} C_VEL
LIN {X 0,Y 463.504,Z 379.217,A -85,B 0,C 180,E1 -8153.951,E2 -8153.951} C_VEL
LIN {X 0,Y 463.128,Z 392.068,A -85,B 0,C 180,E1 -8154.52,E2 -8154.52} C_VEL
LIN {X 0,Y 462.56,Z 404.494,A -85,B 0,C 180,E1 -8155.274,E2 -8155.274} C_VEL
LIN {X 0,Y 462.013,Z 415.636,A -85,B 0,C 180,E1 -8156.145,E2 -8156.145} C_VEL
LIN {X 0,Y 461.504,Z 425.108,A -85,B 0,C 180,E1 -8157.062,E2 -8157.062} C_VEL
LIN {X 0,Y 460.972,Z 435.033,A -85,B 0,C 180,E1 -8158.25,E2 -8158.25} C_VEL
LIN {X 0,Y 460.523,Z 443.527,A -85,B 0,C 180,E1 -8159.509,E2 -8159.509} C_VEL
LIN {X 0,Y 460.238,Z 449.28,A -85,B 0,C 180,E1 -8160.542,E2 -8160.542} C_VEL
LIN {X 0,Y 459.482,Z 452.382,A -85,B 0,C 180,E1 -8161.165,E2 -8161.165} C_VEL
LIN {X 0,Y 456.434,Z 456.955,A -85,B 0,C 180,E1 -8162.199,E2 -8162.199} C_VEL
LIN {X 0,Y 453.365,Z 460.85,A -85,B 0,C 180,E1 -8163.285,E2 -8163.285} C_VEL
LIN {X 0,Y 452.589,Z 462.825,A -85,B 0,C 180,E1 -8163.984,E2 -8163.984} C_VEL
LIN {X 0,Y 452.424,Z 465.612,A -85,B 0,C 180,E1 -8165.204,E2 -8165.204} C_VEL
LIN {X 0,Y 452.323,Z 467.588,A -85,B 0,C 180,E1 -8166.437,E2 -8166.437} C_VEL
LIN {X 0,Y 452.256,Z 469.032,A -85,B 0,C 180,E1 -8168.104,E2 -8168.104} C_VEL
LIN {X 0,Y 452.32,Z 469.24,A -85,B 0,C 180,E1 -8169.063,E2 -8169.063} C_VEL
LIN {X 0,Y 452.308,Z 468.96,A -85,B 0,C 180,E1 -8170.013,E2 -8170.013} C_VEL
LIN {X 0,Y 452.366,Z 467.805,A -85,B 0,C 180,E1 -8171.37,E2 -8171.37} C_VEL
LIN {X 0,Y 452.408,Z 465.493,A -85,B 0,C 180,E1 -8172.835,E2 -8172.835} C_VEL
LIN {X 0,Y 452.595,Z 462.035,A -85,B 0,C 180,E1 -8174.292,E2 -8174.292} C_VEL
LIN {X 0,Y 452.732,Z 457.791,A -85,B 0,C 180,E1 -8175.62,E2 -8175.62} C_VEL
LIN {X 0,Y 452.982,Z 452.144,A -85,B 0,C 180,E1 -8177.001,E2 -8177.001} C_VEL
LIN {X 0,Y 453.307,Z 445.095,A -85,B 0,C 180,E1 -8178.374,E2 -8178.374} C_VEL
LIN {X 0,Y 453.78,Z 436.234,A -85,B 0,C 180,E1 -8179.742,E2 -8179.742} C_VEL
LIN {X 0,Y 454.328,Z 426.162,A -85,B 0,C 180,E1 -8180.991,E2 -8180.991} C_VEL
LIN {X 0,Y 454.874,Z 415.893,A -85,B 0,C 180,E1 -8182.008,E2 -8182.008} C_VEL
LIN {X 0,Y 455.466,Z 404.456,A -85,B 0,C 180,E1 -8182.911,E2 -8182.911} C_VEL
LIN {X 0,Y 456.001,Z 392.59,A -85,B 0,C 180,E1 -8183.641,E2 -8183.641} C_VEL
LIN {X 0,Y 456.398,Z 380.346,A -85,B 0,C 180,E1 -8184.202,E2 -8184.202} C_VEL
LIN {X 0,Y 456.717,Z 367.855,A -85,B 0,C 180,E1 -8184.593,E2 -8184.593} C_VEL
LIN {X 0,Y 456.914,Z 347.705,A -85,B 0,C 180,E1 -8184.955,E2 -8184.955} C_VEL
LIN {X 0,Y 457.466,Z 275.202,A -85,B 0,C 180,E1 -8186.106,E2 -8186.106} C_VEL
LIN {X 0,Y 454.503,Z 258.382,A -85,B 0,C 180,E1 -8186.511,E2 -8186.511} C_VEL
LIN {X 0,Y 454.585,Z 255.089,A -85,B 0,C 180,E1 -8187.121,E2 -8187.121} C_VEL
LIN {X 0,Y 455.246,Z 241.171,A -85,B 0,C 180,E1 -8190.001,E2 -8190.001} C_VEL
LIN {X 0,Y 454.845,Z 237.046,A -85,B 0,C 180,E1 -8190.887,E2 -8190.887} C_VEL
LIN {X 0,Y 453.699,Z 230.633,A -85,B 0,C 180,E1 -8192.332,E2 -8192.332} C_VEL
LIN {X 0,Y 453.629,Z 230.478,A -85,B 0,C 180,E1 -8196.227,E2 -8196.227} C_VEL
LIN {X 0,Y 453.55,Z 230.485,A -85,B 0,C 180,E1 -8198.916,E2 -8198.916} C_VEL
LIN {X 0,Y 453.562,Z 230.482,A -85,B 0,C 180,E1 -8202.553,E2 -8202.553} C_VEL
LIN {X 0,Y 453.506,Z 230.492,A -85,B 0,C 180,E1 -8206.199,E2 -8206.199} C_VEL
LIN {X 0,Y 453.481,Z 230.492,A -85,B 0,C 180,E1 -8209.043,E2 -8209.043} C_VEL
LIN {X 0,Y 453.439,Z 230.505,A -85,B 0,C 180,E1 -8211.839,E2 -8211.839} C_VEL
LIN {X 0,Y 453.458,Z 230.496,A -85,B 0,C 180,E1 -8214.739,E2 -8214.739} C_VEL
LIN {X 0,Y 453.456,Z 230.501,A -85,B 0,C 180,E1 -8217.953,E2 -8217.953} C_VEL
LIN {X 0,Y 453.443,Z 230.499,A -85,B 0,C 180,E1 -8220.763,E2 -8220.763} C_VEL
LIN {X 0,Y 453.434,Z 230.501,A -85,B 0,C 180,E1 -8223.918,E2 -8223.918} C_VEL
LIN {X 0,Y 453.409,Z 230.502,A -85,B 0,C 180,E1 -8227.195,E2 -8227.195} C_VEL
LIN {X 0,Y 453.443,Z 230.505,A -85,B 0,C 180,E1 -8230.616,E2 -8230.616} C_VEL
LIN {X 0,Y 453.434,Z 230.501,A -85,B 0,C 180,E1 -8234.226,E2 -8234.226} C_VEL
LIN {X 0,Y 453.415,Z 230.505,A -85,B 0,C 180,E1 -8237.006,E2 -8237.006} C_VEL
LIN {X 0,Y 453.451,Z 230.497,A -85,B 0,C 180,E1 -8239.417,E2 -8239.417} C_VEL
LIN {X 0,Y 453.434,Z 230.505,A -85,B 0,C 180,E1 -8242.815,E2 -8242.815} C_VEL
LIN {X 0,Y 453.452,Z 230.496,A -85,B 0,C 180,E1 -8246.091,E2 -8246.091} C_VEL
LIN {X 0,Y 453.444,Z 230.504,A -85,B 0,C 180,E1 -8249.243,E2 -8249.243} C_VEL
LIN {X 0,Y 453.463,Z 230.494,A -85,B 0,C 180,E1 -8252.298,E2 -8252.298} C_VEL
LIN {X 0,Y 453.455,Z 230.503,A -85,B 0,C 180,E1 -8255.267,E2 -8255.267} C_VEL
LIN {X 0,Y 453.475,Z 230.493,A -85,B 0,C 180,E1 -8258.42,E2 -8258.42} C_VEL
LIN {X 0,Y 453.519,Z 230.489,A -85,B 0,C 180,E1 -8261.013,E2 -8261.013} C_VEL
LIN {X 0,Y 453.536,Z 230.49,A -85,B 0,C 180,E1 -8263.898,E2 -8263.898} C_VEL
LIN {X 0,Y 453.564,Z 230.486,A -85,B 0,C 180,E1 -8267.475,E2 -8267.475} C_VEL
LIN {X 0,Y 453.562,Z 230.482,A -85,B 0,C 180,E1 -8271.09,E2 -8271.09} C_VEL
LIN {X 0,Y 453.638,Z 230.479,A -85,B 0,C 180,E1 -8273.778,E2 -8273.778} C_VEL
LIN {X 0,Y 453.708,Z 230.464,A -85,B 0,C 180,E1 -8277.34,E2 -8277.34} C_VEL
LIN {X 0,Y 453.772,Z 230.462,A -85,B 0,C 180,E1 -8280.003,E2 -8280.003} C_VEL
LIN {X 0,Y 453.708,Z 230.467,A -85,B 0,C 180,E1 -8282.667,E2 -8282.667} C_VEL
LIN {X 0,Y 453.644,Z 230.479,A -85,B 0,C 180,E1 -8286.229,E2 -8286.229} C_VEL
LIN {X 0,Y 453.57,Z 230.484,A -85,B 0,C 180,E1 -8288.917,E2 -8288.917} C_VEL
LIN {X 0,Y 453.576,Z 230.489,A -85,B 0,C 180,E1 -8292.531,E2 -8292.531} C_VEL
LIN {X 0,Y 453.558,Z 230.485,A -85,B 0,C 180,E1 -8296.198,E2 -8296.198} C_VEL
LIN {X 0,Y 453.53,Z 230.491,A -85,B 0,C 180,E1 -8299.041,E2 -8299.041} C_VEL
LIN {X 0,Y 453.489,Z 230.491,A -85,B 0,C 180,E1 -8301.838,E2 -8301.838} C_VEL
LIN {X 0,Y 453.5,Z 230.495,A -85,B 0,C 180,E1 -8304.738,E2 -8304.738} C_VEL
LIN {X 0,Y 453.477,Z 230.493,A -85,B 0,C 180,E1 -8307.944,E2 -8307.944} C_VEL
LIN {X 0,Y 453.471,Z 230.497,A -85,B 0,C 180,E1 -8310.763,E2 -8310.763} C_VEL
LIN {X 0,Y 453.481,Z 230.493,A -85,B 0,C 180,E1 -8313.915,E2 -8313.915} C_VEL
LIN {X 0,Y 453.463,Z 230.5,A -85,B 0,C 180,E1 -8317.191,E2 -8317.191} C_VEL
LIN {X 0,Y 453.485,Z 230.492,A -85,B 0,C 180,E1 -8320.612,E2 -8320.612} C_VEL
LIN {X 0,Y 453.495,Z 230.49,A -85,B 0,C 180,E1 -8324.529,E2 -8324.529} C_VEL
LIN {X 0,Y 453.45,Z 230.5,A -85,B 0,C 180,E1 -8328.072,E2 -8328.072} C_VEL
LIN {X 0,Y 453.461,Z 230.495,A -85,B 0,C 180,E1 -8330.801,E2 -8330.801} C_VEL
LIN {X 0,Y 453.465,Z 230.503,A -85,B 0,C 180,E1 -8333.917,E2 -8333.917} C_VEL
LIN {X 0,Y 453.496,Z 230.49,A -85,B 0,C 180,E1 -8337.151,E2 -8337.151} C_VEL
LIN {X 0,Y 453.48,Z 230.5,A -85,B 0,C 180,E1 -8340.267,E2 -8340.267} C_VEL
LIN {X 0,Y 453.484,Z 230.497,A -85,B 0,C 180,E1 -8343.291,E2 -8343.291} C_VEL
LIN {X 0,Y 453.531,Z 230.596,A -85,B 0,C 180,E1 -8344.776,E2 -8344.776} C_VEL
LIN {X 0,Y 455.576,Z 241.45,A -85,B 0,C 180,E1 -8347.074,E2 -8347.074} C_VEL
LIN {X 0,Y 455.297,Z 249.966,A -85,B 0,C 180,E1 -8348.73,E2 -8348.73} C_VEL
LIN {X 0,Y 454.614,Z 264.513,A -85,B 0,C 180,E1 -8351.522,E2 -8351.522} C_VEL
LIN {X 0,Y 454.415,Z 270.024,A -85,B 0,C 180,E1 -8352.516,E2 -8352.516} C_VEL
LIN {X 0,Y 457.526,Z 289.417,A -85,B 0,C 180,E1 -8352.968,E2 -8352.968} C_VEL
LIN {X 0,Y 456.691,Z 378.379,A -85,B 0,C 180,E1 -8354.404,E2 -8354.404} C_VEL
LIN {X 0,Y 456.293,Z 392.153,A -85,B 0,C 180,E1 -8354.819,E2 -8354.819} C_VEL
LIN {X 0,Y 455.859,Z 404.53,A -85,B 0,C 180,E1 -8355.376,E2 -8355.376} C_VEL
LIN {X 0,Y 455.352,Z 415.6,A -85,B 0,C 180,E1 -8356.044,E2 -8356.044} C_VEL
LIN {X 0,Y 454.815,Z 427.24,A -85,B 0,C 180,E1 -8356.944,E2 -8356.944} C_VEL
LIN {X 0,Y 454.288,Z 437.571,A -85,B 0,C 180,E1 -8357.944,E2 -8357.944} C_VEL
LIN {X 0,Y 453.741,Z 446.916,A -85,B 0,C 180,E1 -8359.061,E2 -8359.061} C_VEL
LIN {X 0,Y 453.257,Z 455.96,A -85,B 0,C 180,E1 -8360.404,E2 -8360.404} C_VEL
LIN {X 0,Y 452.949,Z 463.244,A -85,B 0,C 180,E1 -8361.747,E2 -8361.747} C_VEL
LIN {X 0,Y 452.729,Z 468.163,A -85,B 0,C 180,E1 -8362.865,E2 -8362.865} C_VEL
LIN {X 0,Y 452.594,Z 472.939,A -85,B 0,C 180,E1 -8364.206,E2 -8364.206} C_VEL
LIN {X 0,Y 452.491,Z 476.591,A -85,B 0,C 180,E1 -8365.545,E2 -8365.545} C_VEL
LIN {X 0,Y 452.458,Z 478.479,A -85,B 0,C 180,E1 -8366.436,E2 -8366.436} C_VEL
LIN {X 0,Y 452.494,Z 479.904,A -85,B 0,C 180,E1 -8367.328,E2 -8367.328} C_VEL
LIN {X 0,Y 452.406,Z 481.537,A -85,B 0,C 180,E1 -8369.109,E2 -8369.109} C_VEL
LIN {X 0,Y 452.41,Z 481.773,A -85,B 0,C 180,E1 -8369.999,E2 -8369.999} C_VEL
LIN {X 0,Y 452.406,Z 481.582,A -85,B 0,C 180,E1 -8370.889,E2 -8370.889} C_VEL
LIN {X 0,Y 452.493,Z 480.01,A -85,B 0,C 180,E1 -8372.669,E2 -8372.669} C_VEL
LIN {X 0,Y 452.458,Z 478.634,A -85,B 0,C 180,E1 -8373.561,E2 -8373.561} C_VEL
LIN {X 0,Y 452.557,Z 475.731,A -85,B 0,C 180,E1 -8374.898,E2 -8374.898} C_VEL
LIN {X 0,Y 452.637,Z 471.199,A -85,B 0,C 180,E1 -8376.417,E2 -8376.417} C_VEL
LIN {X 0,Y 452.904,Z 464.749,A -85,B 0,C 180,E1 -8378.027,E2 -8378.027} C_VEL
LIN {X 0,Y 453.234,Z 457.909,A -85,B 0,C 180,E1 -8379.369,E2 -8379.369} C_VEL
LIN {X 0,Y 453.68,Z 449.38,A -85,B 0,C 180,E1 -8380.712,E2 -8380.712} C_VEL
LIN {X 0,Y 454.269,Z 440.62,A -85,B 0,C 180,E1 -8381.827,E2 -8381.827} C_VEL
LIN {X 0,Y 454.853,Z 430.98,A -85,B 0,C 180,E1 -8382.835,E2 -8382.835} C_VEL
LIN {X 0,Y 455.309,Z 420.54,A -85,B 0,C 180,E1 -8383.727,E2 -8383.727} C_VEL
LIN {X 0,Y 455.877,Z 408.973,A -85,B 0,C 180,E1 -8384.507,E2 -8384.507} C_VEL
LIN {X 0,Y 456.453,Z 396.969,A -85,B 0,C 180,E1 -8385.115,E2 -8385.115} C_VEL
LIN {X 0,Y 456.855,Z 383.981,A -85,B 0,C 180,E1 -8385.587,E2 -8385.587} C_VEL
LIN {X 0,Y 457.156,Z 371.751,A -85,B 0,C 180,E1 -8385.863,E2 -8385.863} C_VEL
LIN {X 0,Y 457.744,Z 288.56,A -85,B 0,C 180,E1 -8387.199,E2 -8387.199} C_VEL
LIN {X 0,Y 454.569,Z 269.923,A -85,B 0,C 180,E1 -8387.665,E2 -8387.665} C_VEL
LIN {X 0,Y 454.655,Z 266.56,A -85,B 0,C 180,E1 -8388.24,E2 -8388.24} C_VEL
LIN {X 0,Y 455.562,Z 248.386,A -85,B 0,C 180,E1 -8391.729,E2 -8391.729} C_VEL
LIN {X 0,Y 455.782,Z 242.333,A -85,B 0,C 180,E1 -8392.912,E2 -8392.912} C_VEL
LIN {X 0,Y 453.594,Z 230.907,A -85,B 0,C 180,E1 -8395.34,E2 -8395.34} C_VEL
LIN {X 0,Y 453.522,Z 230.496,A -85,B 0,C 180,E1 -8395.591,E2 -8395.591} C_VEL
LIN {X 0,Y 453.51,Z 230.492,A -85,B 0,C 180,E1 -8398.71,E2 -8398.71} C_VEL
LIN {X 0,Y 453.466,Z 230.502,A -85,B 0,C 180,E1 -8401.797,E2 -8401.797} C_VEL
LIN {X 0,Y 453.481,Z 230.492,A -85,B 0,C 180,E1 -8404.987,E2 -8404.987} C_VEL
LIN {X 0,Y 453.458,Z 230.496,A -85,B 0,C 180,E1 -8408.31,E2 -8408.31} C_VEL
LIN {X 0,Y 453.494,Z 230.493,A -85,B 0,C 180,E1 -8410.607,E2 -8410.607} C_VEL
LIN {X 0,Y 453.46,Z 230.503,A -85,B 0,C 180,E1 -8414.219,E2 -8414.219} C_VEL
LIN {X 0,Y 453.447,Z 230.492,A -85,B 0,C 180,E1 -8417.001,E2 -8417.001} C_VEL
LIN {X 0,Y 453.47,Z 230.496,A -85,B 0,C 180,E1 -8419.41,E2 -8419.41} C_VEL
LIN {X 0,Y 453.447,Z 230.5,A -85,B 0,C 180,E1 -8422.807,E2 -8422.807} C_VEL
LIN {X 0,Y 453.473,Z 230.497,A -85,B 0,C 180,E1 -8426.084,E2 -8426.084} C_VEL
LIN {X 0,Y 453.471,Z 230.496,A -85,B 0,C 180,E1 -8429.237,E2 -8429.237} C_VEL
LIN {X 0,Y 453.502,Z 230.492,A -85,B 0,C 180,E1 -8432.293,E2 -8432.293} C_VEL
LIN {X 0,Y 453.464,Z 230.497,A -85,B 0,C 180,E1 -8435.26,E2 -8435.26} C_VEL
LIN {X 0,Y 453.474,Z 230.495,A -85,B 0,C 180,E1 -8438.412,E2 -8438.412} C_VEL
LIN {X 0,Y 453.516,Z 230.497,A -85,B 0,C 180,E1 -8441.005,E2 -8441.005} C_VEL
LIN {X 0,Y 453.561,Z 230.481,A -85,B 0,C 180,E1 -8443.877,E2 -8443.877} C_VEL
LIN {X 0,Y 453.555,Z 230.483,A -85,B 0,C 180,E1 -8447.468,E2 -8447.468} C_VEL
LIN {X 0,Y 453.558,Z 230.49,A -85,B 0,C 180,E1 -8451.083,E2 -8451.083} C_VEL
LIN {X 0,Y 453.642,Z 230.476,A -85,B 0,C 180,E1 -8453.771,E2 -8453.771} C_VEL
LIN {X 0,Y 453.686,Z 230.468,A -85,B 0,C 180,E1 -8457.333,E2 -8457.333} C_VEL
LIN {X 0,Y 453.729,Z 230.462,A -85,B 0,C 180,E1 -8459.997,E2 -8459.997} C_VEL
LIN {X 0,Y 453.688,Z 230.467,A -85,B 0,C 180,E1 -8462.66,E2 -8462.66} C_VEL
LIN {X 0,Y 453.616,Z 230.478,A -85,B 0,C 180,E1 -8466.222,E2 -8466.222} C_VEL
LIN {X 0,Y 453.564,Z 230.481,A -85,B 0,C 180,E1 -8468.91,E2 -8468.91} C_VEL
LIN {X 0,Y 453.543,Z 230.484,A -85,B 0,C 180,E1 -8472.525,E2 -8472.525} C_VEL
LIN {X 0,Y 453.521,Z 230.49,A -85,B 0,C 180,E1 -8476.193,E2 -8476.193} C_VEL
LIN {X 0,Y 453.492,Z 230.492,A -85,B 0,C 180,E1 -8479.036,E2 -8479.036} C_VEL
LIN {X 0,Y 453.45,Z 230.502,A -85,B 0,C 180,E1 -8481.833,E2 -8481.833} C_VEL
LIN {X 0,Y 453.472,Z 230.495,A -85,B 0,C 180,E1 -8484.732,E2 -8484.732} C_VEL
LIN {X 0,Y 453.503,Z 230.493,A -85,B 0,C 180,E1 -8487.956,E2 -8487.956} C_VEL
LIN {X 0,Y 453.434,Z 230.5,A -85,B 0,C 180,E1 -8491.522,E2 -8491.522} C_VEL
LIN {X 0,Y 453.457,Z 230.499,A -85,B 0,C 180,E1 -8494.775,E2 -8494.775} C_VEL
LIN {X 0,Y 453.451,Z 230.5,A -85,B 0,C 180,E1 -8498.307,E2 -8498.307} C_VEL
LIN {X 0,Y 453.481,Z 230.497,A -85,B 0,C 180,E1 -8500.604,E2 -8500.604} C_VEL
LIN {X 0,Y 453.445,Z 230.502,A -85,B 0,C 180,E1 -8503.245,E2 -8503.245} C_VEL
LIN {X 0,Y 453.502,Z 230.66,A -85,B 0,C 180,E1 -8505.786,E2 -8505.786} C_VEL
LIN {X 0,Y 455.246,Z 239.933,A -85,B 0,C 180,E1 -8507.81,E2 -8507.81} C_VEL
LIN {X 0,Y 454.699,Z 254.326,A -85,B 0,C 180,E1 -8510.678,E2 -8510.678} C_VEL
LIN {X 0,Y 454.637,Z 258.265,A -85,B 0,C 180,E1 -8511.388,E2 -8511.388} C_VEL
LIN {X 0,Y 457.912,Z 275.502,A -85,B 0,C 180,E1 -8511.833,E2 -8511.833} C_VEL
LIN {X 0,Y 457.053,Z 366.137,A -85,B 0,C 180,E1 -8513.309,E2 -8513.309} C_VEL
LIN {X 0,Y 456.657,Z 380.126,A -85,B 0,C 180,E1 -8513.735,E2 -8513.735} C_VEL
LIN {X 0,Y 456.293,Z 391.978,A -85,B 0,C 180,E1 -8514.272,E2 -8514.272} C_VEL
LIN {X 0,Y 455.729,Z 403.642,A -85,B 0,C 180,E1 -8514.98,E2 -8514.98} C_VEL
LIN {X 0,Y 455.142,Z 414.593,A -85,B 0,C 180,E1 -8515.83,E2 -8515.83} C_VEL
LIN {X 0,Y 454.6,Z 424.689,A -85,B 0,C 180,E1 -8516.806,E2 -8516.806} C_VEL
LIN {X 0,Y 454.055,Z 434.557,A -85,B 0,C 180,E1 -8517.988,E2 -8517.988} C_VEL
LIN {X 0,Y 453.559,Z 443.043,A -85,B 0,C 180,E1 -8519.249,E2 -8519.249} C_VEL
LIN {X 0,Y 453.187,Z 449.97,A -85,B 0,C 180,E1 -8520.513,E2 -8520.513} C_VEL
LIN {X 0,Y 452.922,Z 455.512,A -85,B 0,C 180,E1 -8521.756,E2 -8521.756} C_VEL
LIN {X 0,Y 452.692,Z 460.76,A -85,B 0,C 180,E1 -8523.244,E2 -8523.244} C_VEL
LIN {X 0,Y 452.589,Z 462.825,A -85,B 0,C 180,E1 -8523.984,E2 -8523.984} C_VEL
LIN {X 0,Y 451.828,Z 464.6,A -85,B 0,C 180,E1 -8524.692,E2 -8524.692} C_VEL
LIN {X 0,Y 448.831,Z 466.96,A -85,B 0,C 180,E1 -8525.859,E2 -8525.859} C_VEL
LIN {X 0,Y 446.335,Z 468.268,A -85,B 0,C 180,E1 -8526.815,E2 -8526.815} C_VEL
LIN {X 0,Y 445.258,Z 468.867,A -85,B 0,C 180,E1 -8527.561,E2 -8527.561} C_VEL
LIN {X 0,Y 445.167,Z 468.984,A -85,B 0,C 180,E1 -8527.816,E2 -8527.816} C_VEL
LIN {X 0,Y 445.192,Z 469.304,A -85,B 0,C 180,E1 -8528.712,E2 -8528.712} C_VEL
LIN {X 0,Y 445.204,Z 469.222,A -85,B 0,C 180,E1 -8529.68,E2 -8529.68} C_VEL
LIN {X 0,Y 445.264,Z 468.077,A -85,B 0,C 180,E1 -8531.251,E2 -8531.251} C_VEL
LIN {X 0,Y 445.283,Z 466.217,A -85,B 0,C 180,E1 -8532.551,E2 -8532.551} C_VEL
LIN {X 0,Y 445.495,Z 462.564,A -85,B 0,C 180,E1 -8534.2,E2 -8534.2} C_VEL
LIN {X 0,Y 445.694,Z 457.362,A -85,B 0,C 180,E1 -8535.854,E2 -8535.854} C_VEL
LIN {X 0,Y 445.931,Z 451.596,A -85,B 0,C 180,E1 -8537.255,E2 -8537.255} C_VEL
LIN {X 0,Y 446.337,Z 444.335,A -85,B 0,C 180,E1 -8538.65,E2 -8538.65} C_VEL
LIN {X 0,Y 446.859,Z 435.277,A -85,B 0,C 180,E1 -8540.039,E2 -8540.039} C_VEL
LIN {X 0,Y 447.36,Z 426.158,A -85,B 0,C 180,E1 -8541.172,E2 -8541.172} C_VEL
LIN {X 0,Y 447.968,Z 415.631,A -85,B 0,C 180,E1 -8542.225,E2 -8542.225} C_VEL
LIN {X 0,Y 448.565,Z 404.128,A -85,B 0,C 180,E1 -8543.14,E2 -8543.14} C_VEL
LIN {X 0,Y 449.125,Z 392.139,A -85,B 0,C 180,E1 -8543.882,E2 -8543.882} C_VEL
LIN {X 0,Y 449.523,Z 379.649,A -85,B 0,C 180,E1 -8544.45,E2 -8544.45} C_VEL
LIN {X 0,Y 449.913,Z 366.67,A -85,B 0,C 180,E1 -8544.848,E2 -8544.848} C_VEL
LIN {X 0,Y 450.292,Z 324.843,A -85,B 0,C 180,E1 -8545.552,E2 -8545.552} C_VEL
LIN {X 0,Y 450.587,Z 275.783,A -85,B 0,C 180,E1 -8546.344,E2 -8546.344} C_VEL
LIN {X 0,Y 447.524,Z 258.552,A -85,B 0,C 180,E1 -8546.766,E2 -8546.766} C_VEL
LIN {X 0,Y 447.627,Z 255.594,A -85,B 0,C 180,E1 -8547.302,E2 -8547.302} C_VEL
LIN {X 0,Y 448.287,Z 241.661,A -85,B 0,C 180,E1 -8550.226,E2 -8550.226} C_VEL
LIN {X 0,Y 446.857,Z 232.545,A -85,B 0,C 180,E1 -8552.255,E2 -8552.255} C_VEL
LIN {X 0,Y 446.682,Z 231.373,A -85,B 0,C 180,E1 -8552.594,E2 -8552.594} C_VEL
LIN {X 0,Y 446.598,Z 231.353,A -85,B 0,C 180,E1 -8556.326,E2 -8556.326} C_VEL
LIN {X 0,Y 446.496,Z 231.365,A -85,B 0,C 180,E1 -8559.058,E2 -8559.058} C_VEL
LIN {X 0,Y 446.493,Z 231.363,A -85,B 0,C 180,E1 -8562.732,E2 -8562.732} C_VEL
LIN {X 0,Y 446.451,Z 231.369,A -85,B 0,C 180,E1 -8566.462,E2 -8566.462} C_VEL
LIN {X 0,Y 446.431,Z 231.372,A -85,B 0,C 180,E1 -8569.306,E2 -8569.306} C_VEL
LIN {X 0,Y 446.38,Z 231.382,A -85,B 0,C 180,E1 -8572.203,E2 -8572.203} C_VEL
LIN {X 0,Y 446.402,Z 231.374,A -85,B 0,C 180,E1 -8575.157,E2 -8575.157} C_VEL
LIN {X 0,Y 446.407,Z 231.382,A -85,B 0,C 180,E1 -8578.185,E2 -8578.185} C_VEL
LIN {X 0,Y 446.382,Z 231.376,A -85,B 0,C 180,E1 -8581.304,E2 -8581.304} C_VEL
LIN {X 0,Y 446.39,Z 231.382,A -85,B 0,C 180,E1 -8584.528,E2 -8584.528} C_VEL
LIN {X 0,Y 446.37,Z 231.381,A -85,B 0,C 180,E1 -8588.08,E2 -8588.08} C_VEL
LIN {X 0,Y 446.376,Z 231.377,A -85,B 0,C 180,E1 -8591.398,E2 -8591.398} C_VEL
LIN {X 0,Y 446.398,Z 231.377,A -85,B 0,C 180,E1 -8595.112,E2 -8595.112} C_VEL
LIN {X 0,Y 446.386,Z 231.382,A -85,B 0,C 180,E1 -8598.611,E2 -8598.611} C_VEL
LIN {X 0,Y 446.393,Z 231.375,A -85,B 0,C 180,E1 -8601.926,E2 -8601.926} C_VEL
LIN {X 0,Y 446.407,Z 231.376,A -85,B 0,C 180,E1 -8605.481,E2 -8605.481} C_VEL
LIN {X 0,Y 446.394,Z 231.378,A -85,B 0,C 180,E1 -8608.703,E2 -8608.703} C_VEL
LIN {X 0,Y 446.413,Z 231.374,A -85,B 0,C 180,E1 -8611.841,E2 -8611.841} C_VEL
LIN {X 0,Y 446.405,Z 231.376,A -85,B 0,C 180,E1 -8614.849,E2 -8614.849} C_VEL
LIN {X 0,Y 446.442,Z 231.369,A -85,B 0,C 180,E1 -8618.25,E2 -8618.25} C_VEL
LIN {X 0,Y 446.445,Z 231.376,A -85,B 0,C 180,E1 -8621.653,E2 -8621.653} C_VEL
LIN {X 0,Y 446.492,Z 231.363,A -85,B 0,C 180,E1 -8624.483,E2 -8624.483} C_VEL
LIN {X 0,Y 446.506,Z 231.364,A -85,B 0,C 180,E1 -8628.197,E2 -8628.197} C_VEL
LIN {X 0,Y 446.513,Z 231.36,A -85,B 0,C 180,E1 -8630.948,E2 -8630.948} C_VEL
LIN {X 0,Y 446.608,Z 231.353,A -85,B 0,C 180,E1 -8633.68,E2 -8633.68} C_VEL
LIN {X 0,Y 446.657,Z 231.343,A -85,B 0,C 180,E1 -8637.298,E2 -8637.298} C_VEL
LIN {X 0,Y 446.723,Z 231.34,A -85,B 0,C 180,E1 -8640.003,E2 -8640.003} C_VEL
LIN {X 0,Y 446.658,Z 231.345,A -85,B 0,C 180,E1 -8642.709,E2 -8642.709} C_VEL
LIN {X 0,Y 446.614,Z 231.356,A -85,B 0,C 180,E1 -8646.327,E2 -8646.327} C_VEL
LIN {X 0,Y 446.521,Z 231.36,A -85,B 0,C 180,E1 -8649.059,E2 -8649.059} C_VEL
LIN {X 0,Y 446.534,Z 231.364,A -85,B 0,C 180,E1 -8652.732,E2 -8652.732} C_VEL
LIN {X 0,Y 446.502,Z 231.367,A -85,B 0,C 180,E1 -8656.462,E2 -8656.462} C_VEL
LIN {X 0,Y 446.482,Z 231.366,A -85,B 0,C 180,E1 -8659.306,E2 -8659.306} C_VEL
LIN {X 0,Y 446.43,Z 231.371,A -85,B 0,C 180,E1 -8662.202,E2 -8662.202} C_VEL
LIN {X 0,Y 446.443,Z 231.375,A -85,B 0,C 180,E1 -8665.156,E2 -8665.156} C_VEL
LIN {X 0,Y 446.431,Z 231.37,A -85,B 0,C 180,E1 -8668.185,E2 -8668.185} C_VEL
LIN {X 0,Y 446.423,Z 231.378,A -85,B 0,C 180,E1 -8671.303,E2 -8671.303} C_VEL
LIN {X 0,Y 446.436,Z 231.37,A -85,B 0,C 180,E1 -8674.525,E2 -8674.525} C_VEL
LIN {X 0,Y 446.425,Z 231.372,A -85,B 0,C 180,E1 -8678.079,E2 -8678.079} C_VEL
LIN {X 0,Y 446.415,Z 231.379,A -85,B 0,C 180,E1 -8681.395,E2 -8681.395} C_VEL
LIN {X 0,Y 446.436,Z 231.372,A -85,B 0,C 180,E1 -8685.108,E2 -8685.108} C_VEL
LIN {X 0,Y 446.414,Z 231.373,A -85,B 0,C 180,E1 -8688.606,E2 -8688.606} C_VEL
LIN {X 0,Y 446.424,Z 231.379,A -85,B 0,C 180,E1 -8691.922,E2 -8691.922} C_VEL
LIN {X 0,Y 446.442,Z 231.371,A -85,B 0,C 180,E1 -8695.477,E2 -8695.477} C_VEL
LIN {X 0,Y 446.429,Z 231.375,A -85,B 0,C 180,E1 -8698.699,E2 -8698.699} C_VEL
LIN {X 0,Y 446.463,Z 231.374,A -85,B 0,C 180,E1 -8701.83,E2 -8701.83} C_VEL
LIN {X 0,Y 446.508,Z 231.524,A -85,B 0,C 180,E1 -8704.6,E2 -8704.6} C_VEL
LIN {X 0,Y 448.557,Z 242.427,A -85,B 0,C 180,E1 -8706.938,E2 -8706.938} C_VEL
LIN {X 0,Y 448.401,Z 249.736,A -85,B 0,C 180,E1 -8708.386,E2 -8708.386} C_VEL
LIN {X 0,Y 447.692,Z 264.286,A -85,B 0,C 180,E1 -8711.226,E2 -8711.226} C_VEL
LIN {X 0,Y 447.425,Z 269.736,A -85,B 0,C 180,E1 -8712.236,E2 -8712.236} C_VEL
LIN {X 0,Y 448.102,Z 274.167,A -85,B 0,C 180,E1 -8712.385,E2 -8712.385} C_VEL
LIN {X 0,Y 450.699,Z 290.191,A -85,B 0,C 180,E1 -8712.741,E2 -8712.741} C_VEL
LIN {X 0,Y 449.845,Z 377.536,A -85,B 0,C 180,E1 -8714.161,E2 -8714.161} C_VEL
LIN {X 0,Y 449.48,Z 390.793,A -85,B 0,C 180,E1 -8714.555,E2 -8714.555} C_VEL
LIN {X 0,Y 448.965,Z 404.083,A -85,B 0,C 180,E1 -8715.146,E2 -8715.146} C_VEL
LIN {X 0,Y 448.437,Z 415.24,A -85,B 0,C 180,E1 -8715.824,E2 -8715.824} C_VEL
LIN {X 0,Y 447.886,Z 426.929,A -85,B 0,C 180,E1 -8716.739,E2 -8716.739} C_VEL
LIN {X 0,Y 447.323,Z 437.297,A -85,B 0,C 180,E1 -8717.753,E2 -8717.753} C_VEL
LIN {X 0,Y 446.736,Z 446.684,A -85,B 0,C 180,E1 -8718.887,E2 -8718.887} C_VEL
LIN {X 0,Y 446.233,Z 455.752,A -85,B 0,C 180,E1 -8720.251,E2 -8720.251} C_VEL
LIN {X 0,Y 445.885,Z 463.056,A -85,B 0,C 180,E1 -8721.615,E2 -8721.615} C_VEL
LIN {X 0,Y 445.676,Z 467.993,A -85,B 0,C 180,E1 -8722.751,E2 -8722.751} C_VEL
LIN {X 0,Y 445.505,Z 472.187,A -85,B 0,C 180,E1 -8723.924,E2 -8723.924} C_VEL
LIN {X 0,Y 445.418,Z 476.452,A -85,B 0,C 180,E1 -8725.474,E2 -8725.474} C_VEL
LIN {X 0,Y 445.358,Z 478.346,A -85,B 0,C 180,E1 -8726.38,E2 -8726.38} C_VEL
LIN {X 0,Y 445.401,Z 479.784,A -85,B 0,C 180,E1 -8727.285,E2 -8727.285} C_VEL
LIN {X 0,Y 445.318,Z 481.429,A -85,B 0,C 180,E1 -8729.094,E2 -8729.094} C_VEL
LIN {X 0,Y 445.319,Z 481.672,A -85,B 0,C 180,E1 -8729.999,E2 -8729.999} C_VEL
LIN {X 0,Y 445.318,Z 481.492,A -85,B 0,C 180,E1 -8730.903,E2 -8730.903} C_VEL
LIN {X 0,Y 445.401,Z 479.931,A -85,B 0,C 180,E1 -8732.712,E2 -8732.712} C_VEL
LIN {X 0,Y 445.358,Z 478.562,A -85,B 0,C 180,E1 -8733.618,E2 -8733.618} C_VEL
LIN {X 0,Y 445.49,Z 475.669,A -85,B 0,C 180,E1 -8734.976,E2 -8734.976} C_VEL
LIN {X 0,Y 445.608,Z 470.345,A -85,B 0,C 180,E1 -8736.746,E2 -8736.746} C_VEL
LIN {X 0,Y 445.862,Z 464.718,A -85,B 0,C 180,E1 -8738.154,E2 -8738.154} C_VEL
LIN {X 0,Y 446.221,Z 457.892,A -85,B 0,C 180,E1 -8739.518,E2 -8739.518} C_VEL
LIN {X 0,Y 446.68,Z 449.389,A -85,B 0,C 180,E1 -8740.882,E2 -8740.882} C_VEL
LIN {X 0,Y 447.307,Z 440.651,A -85,B 0,C 180,E1 -8742.014,E2 -8742.014} C_VEL
LIN {X 0,Y 447.969,Z 430.052,A -85,B 0,C 180,E1 -8743.133,E2 -8743.133} C_VEL
LIN {X 0,Y 448.516,Z 419.18,A -85,B 0,C 180,E1 -8744.055,E2 -8744.055} C_VEL
LIN {X 0,Y 449.11,Z 407.178,A -85,B 0,C 180,E1 -8744.846,E2 -8744.846} C_VEL
LIN {X 0,Y 449.707,Z 394.689,A -85,B 0,C 180,E1 -8745.464,E2 -8745.464} C_VEL
LIN {X 0,Y 450.083,Z 382.667,A -85,B 0,C 180,E1 -8745.886,E2 -8745.886} C_VEL
LIN {X 0,Y 450.425,Z 367.644,A -85,B 0,C 180,E1 -8746.193,E2 -8746.193} C_VEL
LIN {X 0,Y 451.04,Z 289.45,A -85,B 0,C 180,E1 -8747.473,E2 -8747.473} C_VEL
LIN {X 0,Y 447.652,Z 269.746,A -85,B 0,C 180,E1 -8747.979,E2 -8747.979} C_VEL
LIN {X 0,Y 448.019,Z 261.116,A -85,B 0,C 180,E1 -8749.595,E2 -8749.595} C_VEL
LIN {X 0,Y 448.908,Z 245.291,A -85,B 0,C 180,E1 -8752.696,E2 -8752.696} C_VEL
LIN {X 0,Y 447.973,Z 238.774,A -85,B 0,C 180,E1 -8754.071,E2 -8754.071} C_VEL
LIN {X 0,Y 446.505,Z 231.474,A -85,B 0,C 180,E1 -8755.709,E2 -8755.709} C_VEL
LIN {X 0,Y 446.45,Z 231.372,A -85,B 0,C 180,E1 -8759.207,E2 -8759.207} C_VEL
LIN {X 0,Y 446.424,Z 231.373,A -85,B 0,C 180,E1 -8762.359,E2 -8762.359} C_VEL
LIN {X 0,Y 446.419,Z 231.373,A -85,B 0,C 180,E1 -8765.624,E2 -8765.624} C_VEL
LIN {X 0,Y 446.41,Z 231.373,A -85,B 0,C 180,E1 -8769.028,E2 -8769.028} C_VEL
LIN {X 0,Y 446.422,Z 231.371,A -85,B 0,C 180,E1 -8772.273,E2 -8772.273} C_VEL
LIN {X 0,Y 446.422,Z 231.372,A -85,B 0,C 180,E1 -8775.105,E2 -8775.105} C_VEL
LIN {X 0,Y 446.409,Z 231.38,A -85,B 0,C 180,E1 -8778.604,E2 -8778.604} C_VEL
LIN {X 0,Y 446.408,Z 231.376,A -85,B 0,C 180,E1 -8781.919,E2 -8781.919} C_VEL
LIN {X 0,Y 446.425,Z 231.373,A -85,B 0,C 180,E1 -8785.474,E2 -8785.474} C_VEL
LIN {X 0,Y 446.412,Z 231.381,A -85,B 0,C 180,E1 -8788.697,E2 -8788.697} C_VEL
LIN {X 0,Y 446.444,Z 231.369,A -85,B 0,C 180,E1 -8791.827,E2 -8791.827} C_VEL
LIN {X 0,Y 446.416,Z 231.375,A -85,B 0,C 180,E1 -8794.842,E2 -8794.842} C_VEL
LIN {X 0,Y 446.442,Z 231.37,A -85,B 0,C 180,E1 -8798.242,E2 -8798.242} C_VEL
LIN {X 0,Y 446.442,Z 231.37,A -85,B 0,C 180,E1 -8801.646,E2 -8801.646} C_VEL
LIN {X 0,Y 446.496,Z 231.362,A -85,B 0,C 180,E1 -8804.476,E2 -8804.476} C_VEL
LIN {X 0,Y 446.505,Z 231.358,A -85,B 0,C 180,E1 -8808.19,E2 -8808.19} C_VEL
LIN {X 0,Y 446.507,Z 231.366,A -85,B 0,C 180,E1 -8810.941,E2 -8810.941} C_VEL
LIN {X 0,Y 446.611,Z 231.353,A -85,B 0,C 180,E1 -8813.673,E2 -8813.673} C_VEL
LIN {X 0,Y 446.636,Z 231.346,A -85,B 0,C 180,E1 -8817.291,E2 -8817.291} C_VEL
LIN {X 0,Y 446.68,Z 231.34,A -85,B 0,C 180,E1 -8819.997,E2 -8819.997} C_VEL
LIN {X 0,Y 446.638,Z 231.345,A -85,B 0,C 180,E1 -8822.702,E2 -8822.702} C_VEL
LIN {X 0,Y 446.586,Z 231.353,A -85,B 0,C 180,E1 -8826.321,E2 -8826.321} C_VEL
LIN {X 0,Y 446.511,Z 231.361,A -85,B 0,C 180,E1 -8829.052,E2 -8829.052} C_VEL
LIN {X 0,Y 446.5,Z 231.36,A -85,B 0,C 180,E1 -8832.726,E2 -8832.726} C_VEL
LIN {X 0,Y 446.465,Z 231.368,A -85,B 0,C 180,E1 -8836.456,E2 -8836.456} C_VEL
LIN {X 0,Y 446.443,Z 231.37,A -85,B 0,C 180,E1 -8839.3,E2 -8839.3} C_VEL
LIN {X 0,Y 446.392,Z 231.381,A -85,B 0,C 180,E1 -8842.196,E2 -8842.196} C_VEL
LIN {X 0,Y 446.416,Z 231.372,A -85,B 0,C 180,E1 -8845.15,E2 -8845.15} C_VEL
LIN {X 0,Y 446.456,Z 231.368,A -85,B 0,C 180,E1 -8848.175,E2 -8848.175} C_VEL
LIN {X 0,Y 446.388,Z 231.379,A -85,B 0,C 180,E1 -8851.772,E2 -8851.772} C_VEL
LIN {X 0,Y 446.399,Z 231.381,A -85,B 0,C 180,E1 -8854.52,E2 -8854.52} C_VEL
LIN {X 0,Y 446.405,Z 231.378,A -85,B 0,C 180,E1 -8858.08,E2 -8858.08} C_VEL
LIN {X 0,Y 446.412,Z 231.379,A -85,B 0,C 180,E1 -8860.918,E2 -8860.918} C_VEL
LIN {X 0,Y 446.408,Z 231.377,A -85,B 0,C 180,E1 -8863.838,E2 -8863.838} C_VEL
LIN {X 0,Y 446.458,Z 231.6,A -85,B 0,C 180,E1 -8865.553,E2 -8865.553} C_VEL
LIN {X 0,Y 448.26,Z 240.872,A -85,B 0,C 180,E1 -8867.613,E2 -8867.613} C_VEL
LIN {X 0,Y 448.027,Z 249.589,A -85,B 0,C 180,E1 -8869.386,E2 -8869.386} C_VEL
LIN {X 0,Y 447.728,Z 258.113,A -85,B 0,C 180,E1 -8871.055,E2 -8871.055} C_VEL
LIN {X 0,Y 449.524,Z 267.084,A -85,B 0,C 180,E1 -8871.323,E2 -8871.323} C_VEL
LIN {X 0,Y 451.155,Z 275.944,A -85,B 0,C 180,E1 -8871.545,E2 -8871.545} C_VEL
LIN {X 0,Y 450.299,Z 365.928,A -85,B 0,C 180,E1 -8873.037,E2 -8873.037} C_VEL
LIN {X 0,Y 449.894,Z 379.492,A -85,B 0,C 180,E1 -8873.45,E2 -8873.45} C_VEL
LIN {X 0,Y 449.467,Z 391.751,A -85,B 0,C 180,E1 -8874.006,E2 -8874.006} C_VEL
LIN {X 0,Y 448.885,Z 403.683,A -85,B 0,C 180,E1 -8874.739,E2 -8874.739} C_VEL
LIN {X 0,Y 448.243,Z 415.038,A -85,B 0,C 180,E1 -8875.638,E2 -8875.638} C_VEL
LIN {X 0,Y 447.624,Z 425.444,A -85,B 0,C 180,E1 -8876.668,E2 -8876.668} C_VEL
LIN {X 0,Y 447.133,Z 433.93,A -85,B 0,C 180,E1 -8877.698,E2 -8877.698} C_VEL
LIN {X 0,Y 446.588,Z 442.554,A -85,B 0,C 180,E1 -8878.978,E2 -8878.978} C_VEL
LIN {X 0,Y 446.156,Z 450.243,A -85,B 0,C 180,E1 -8880.397,E2 -8880.397} C_VEL
LIN {X 0,Y 445.852,Z 456.23,A -85,B 0,C 180,E1 -8881.78,E2 -8881.78} C_VEL
LIN {X 0,Y 445.593,Z 461.328,A -85,B 0,C 180,E1 -8883.29,E2 -8883.29} C_VEL
LIN {X 0,Y 445.42,Z 465.042,A -85,B 0,C 180,E1 -8884.787,E2 -8884.787} C_VEL
LIN {X 0,Y 445.253,Z 467.542,A -85,B 0,C 180,E1 -8886.261,E2 -8886.261} C_VEL
LIN {X 0,Y 445.167,Z 468.984,A -85,B 0,C 180,E1 -8887.816,E2 -8887.816} C_VEL
LIN {X 0,Y 444.493,Z 469.305,A -85,B 0,C 180,E1 -8888.571,E2 -8888.571} C_VEL
LIN {X 0,Y 441.652,Z 469.219,A -85,B 0,C 180,E1 -8889.8,E2 -8889.8} C_VEL
LIN {X 0,Y 439.264,Z 468.61,A -85,B 0,C 180,E1 -8890.788,E2 -8890.788} C_VEL
LIN {X 0,Y 438.247,Z 467.835,A -85,B 0,C 180,E1 -8891.546,E2 -8891.546} C_VEL
LIN {X 0,Y 438.168,Z 467.458,A -85,B 0,C 180,E1 -8891.801,E2 -8891.801} C_VEL
LIN {X 0,Y 438.272,Z 465.099,A -85,B 0,C 180,E1 -8893.225,E2 -8893.225} C_VEL
LIN {X 0,Y 438.46,Z 461.581,A -85,B 0,C 180,E1 -8894.666,E2 -8894.666} C_VEL
LIN {X 0,Y 438.657,Z 456.933,A -85,B 0,C 180,E1 -8896.096,E2 -8896.096} C_VEL
LIN {X 0,Y 439.014,Z 450.146,A -85,B 0,C 180,E1 -8897.694,E2 -8897.694} C_VEL
LIN {X 0,Y 439.406,Z 442.185,A -85,B 0,C 180,E1 -8899.169,E2 -8899.169} C_VEL
LIN {X 0,Y 439.921,Z 434.328,A -85,B 0,C 180,E1 -8900.345,E2 -8900.345} C_VEL
LIN {X 0,Y 440.496,Z 424.597,A -85,B 0,C 180,E1 -8901.53,E2 -8901.53} C_VEL
LIN {X 0,Y 441.144,Z 414.051,A -85,B 0,C 180,E1 -8902.564,E2 -8902.564} C_VEL
LIN {X 0,Y 441.767,Z 402.126,A -85,B 0,C 180,E1 -8903.493,E2 -8903.493} C_VEL
LIN {X 0,Y 442.304,Z 389.346,A -85,B 0,C 180,E1 -8904.245,E2 -8904.245} C_VEL
LIN {X 0,Y 442.751,Z 376.516,A -85,B 0,C 180,E1 -8904.793,E2 -8904.793} C_VEL
LIN {X 0,Y 443.053,Z 364.106,A -85,B 0,C 180,E1 -8905.139,E2 -8905.139} C_VEL
LIN {X 0,Y 443.83,Z 276.975,A -85,B 0,C 180,E1 -8906.575,E2 -8906.575} C_VEL
LIN {X 0,Y 440.604,Z 258.752,A -85,B 0,C 180,E1 -8907.026,E2 -8907.026} C_VEL
LIN {X 0,Y 440.603,Z 257.181,A -85,B 0,C 180,E1 -8907.259,E2 -8907.259} C_VEL
LIN {X 0,Y 441.313,Z 243.207,A -85,B 0,C 180,E1 -8910.23,E2 -8910.23} C_VEL
LIN {X 0,Y 440.407,Z 237.092,A -85,B 0,C 180,E1 -8911.602,E2 -8911.602} C_VEL
LIN {X 0,Y 439.613,Z 232.29,A -85,B 0,C 180,E1 -8912.75,E2 -8912.75} C_VEL
LIN {X 0,Y 439.573,Z 232.229,A -85,B 0,C 180,E1 -8916.427,E2 -8916.427} C_VEL
LIN {X 0,Y 439.458,Z 232.243,A -85,B 0,C 180,E1 -8919.204,E2 -8919.204} C_VEL
LIN {X 0,Y 439.464,Z 232.238,A -85,B 0,C 180,E1 -8922.729,E2 -8922.729} C_VEL
LIN {X 0,Y 439.408,Z 232.247,A -85,B 0,C 180,E1 -8926.351,E2 -8926.351} C_VEL
LIN {X 0,Y 439.365,Z 232.256,A -85,B 0,C 180,E1 -8929.629,E2 -8929.629} C_VEL
LIN {X 0,Y 439.326,Z 232.257,A -85,B 0,C 180,E1 -8932.579,E2 -8932.579} C_VEL
LIN {X 0,Y 439.34,Z 232.256,A -85,B 0,C 180,E1 -8935.59,E2 -8935.59} C_VEL
LIN {X 0,Y 439.363,Z 232.253,A -85,B 0,C 180,E1 -8938.679,E2 -8938.679} C_VEL
LIN {X 0,Y 439.334,Z 232.26,A -85,B 0,C 180,E1 -8942.033,E2 -8942.033} C_VEL
LIN {X 0,Y 439.358,Z 232.251,A -85,B 0,C 180,E1 -8945.343,E2 -8945.343} C_VEL
LIN {X 0,Y 439.327,Z 232.262,A -85,B 0,C 180,E1 -8948.602,E2 -8948.602} C_VEL
LIN {X 0,Y 439.326,Z 232.259,A -85,B 0,C 180,E1 -8952.214,E2 -8952.214} C_VEL
LIN {X 0,Y 439.353,Z 232.254,A -85,B 0,C 180,E1 -8955.272,E2 -8955.272} C_VEL
LIN {X 0,Y 439.347,Z 232.261,A -85,B 0,C 180,E1 -8958.751,E2 -8958.751} C_VEL
LIN {X 0,Y 439.346,Z 232.254,A -85,B 0,C 180,E1 -8961.614,E2 -8961.614} C_VEL
LIN {X 0,Y 439.38,Z 232.255,A -85,B 0,C 180,E1 -8964.848,E2 -8964.848} C_VEL
LIN {X 0,Y 439.352,Z 232.252,A -85,B 0,C 180,E1 -8968.143,E2 -8968.143} C_VEL
LIN {X 0,Y 439.376,Z 232.253,A -85,B 0,C 180,E1 -8971.614,E2 -8971.614} C_VEL
LIN {X 0,Y 439.353,Z 232.252,A -85,B 0,C 180,E1 -8974.417,E2 -8974.417} C_VEL
LIN {X 0,Y 439.355,Z 232.261,A -85,B 0,C 180,E1 -8977.429,E2 -8977.429} C_VEL
LIN {X 0,Y 439.437,Z 232.242,A -85,B 0,C 180,E1 -8980.668,E2 -8980.668} C_VEL
LIN {X 0,Y 439.452,Z 232.241,A -85,B 0,C 180,E1 -8984.228,E2 -8984.228} C_VEL
LIN {X 0,Y 439.476,Z 232.242,A -85,B 0,C 180,E1 -8988.005,E2 -8988.005} C_VEL
LIN {X 0,Y 439.483,Z 232.242,A -85,B 0,C 180,E1 -8991.729,E2 -8991.729} C_VEL
LIN {X 0,Y 439.599,Z 232.223,A -85,B 0,C 180,E1 -8994.499,E2 -8994.499} C_VEL
LIN {X 0,Y 439.633,Z 232.225,A -85,B 0,C 180,E1 -8998.171,E2 -8998.171} C_VEL
LIN {X 0,Y 439.581,Z 232.224,A -85,B 0,C 180,E1 -9000.92,E2 -9000.92} C_VEL
LIN {X 0,Y 439.609,Z 232.222,A -85,B 0,C 180,E1 -9002.752,E2 -9002.752} C_VEL
LIN {X 0,Y 439.567,Z 232.233,A -85,B 0,C 180,E1 -9006.429,E2 -9006.429} C_VEL
LIN {X 0,Y 439.488,Z 232.236,A -85,B 0,C 180,E1 -9009.205,E2 -9009.205} C_VEL
LIN {X 0,Y 439.477,Z 232.24,A -85,B 0,C 180,E1 -9012.94,E2 -9012.94} C_VEL
LIN {X 0,Y 439.459,Z 232.243,A -85,B 0,C 180,E1 -9016.35,E2 -9016.35} C_VEL
LIN {X 0,Y 439.415,Z 232.245,A -85,B 0,C 180,E1 -9019.629,E2 -9019.629} C_VEL
LIN {X 0,Y 439.376,Z 232.253,A -85,B 0,C 180,E1 -9022.578,E2 -9022.578} C_VEL
LIN {X 0,Y 439.385,Z 232.25,A -85,B 0,C 180,E1 -9025.589,E2 -9025.589} C_VEL
LIN {X 0,Y 439.397,Z 232.25,A -85,B 0,C 180,E1 -9028.678,E2 -9028.678} C_VEL
LIN {X 0,Y 439.377,Z 232.249,A -85,B 0,C 180,E1 -9032.03,E2 -9032.03} C_VEL
LIN {X 0,Y 439.405,Z 232.254,A -85,B 0,C 180,E1 -9035.34,E2 -9035.34} C_VEL
LIN {X 0,Y 439.377,Z 232.249,A -85,B 0,C 180,E1 -9038.598,E2 -9038.598} C_VEL
LIN {X 0,Y 439.363,Z 232.252,A -85,B 0,C 180,E1 -9042.211,E2 -9042.211} C_VEL
LIN {X 0,Y 439.39,Z 232.251,A -85,B 0,C 180,E1 -9045.268,E2 -9045.268} C_VEL
LIN {X 0,Y 439.377,Z 232.249,A -85,B 0,C 180,E1 -9048.748,E2 -9048.748} C_VEL
LIN {X 0,Y 439.378,Z 232.254,A -85,B 0,C 180,E1 -9051.61,E2 -9051.61} C_VEL
LIN {X 0,Y 439.412,Z 232.245,A -85,B 0,C 180,E1 -9054.844,E2 -9054.844} C_VEL
LIN {X 0,Y 439.387,Z 232.256,A -85,B 0,C 180,E1 -9058.139,E2 -9058.139} C_VEL
LIN {X 0,Y 439.418,Z 232.25,A -85,B 0,C 180,E1 -9061.605,E2 -9061.605} C_VEL
LIN {X 0,Y 439.467,Z 232.431,A -85,B 0,C 180,E1 -9064.418,E2 -9064.418} C_VEL
LIN {X 0,Y 441.517,Z 243.331,A -85,B 0,C 180,E1 -9066.783,E2 -9066.783} C_VEL
LIN {X 0,Y 441.614,Z 248.283,A -85,B 0,C 180,E1 -9067.791,E2 -9067.791} C_VEL
LIN {X 0,Y 440.675,Z 265.27,A -85,B 0,C 180,E1 -9071.157,E2 -9071.157} C_VEL
LIN {X 0,Y 440.474,Z 269.629,A -85,B 0,C 180,E1 -9071.973,E2 -9071.973} C_VEL
LIN {X 0,Y 441.042,Z 273.595,A -85,B 0,C 180,E1 -9072.112,E2 -9072.112} C_VEL
LIN {X 0,Y 443.877,Z 291.582,A -85,B 0,C 180,E1 -9072.517,E2 -9072.517} C_VEL
LIN {X 0,Y 442.983,Z 377.725,A -85,B 0,C 180,E1 -9073.938,E2 -9073.938} C_VEL
LIN {X 0,Y 442.596,Z 390.899,A -85,B 0,C 180,E1 -9074.338,E2 -9074.338} C_VEL
LIN {X 0,Y 442.107,Z 403.598,A -85,B 0,C 180,E1 -9074.91,E2 -9074.91} C_VEL
LIN {X 0,Y 441.531,Z 414.878,A -85,B 0,C 180,E1 -9075.598,E2 -9075.598} C_VEL
LIN {X 0,Y 440.936,Z 426.117,A -85,B 0,C 180,E1 -9076.481,E2 -9076.481} C_VEL
LIN {X 0,Y 440.36,Z 437.023,A -85,B 0,C 180,E1 -9077.556,E2 -9077.556} C_VEL
LIN {X 0,Y 439.749,Z 446.452,A -85,B 0,C 180,E1 -9078.709,E2 -9078.709} C_VEL
LIN {X 0,Y 439.222,Z 455.544,A -85,B 0,C 180,E1 -9080.094,E2 -9080.094} C_VEL
LIN {X 0,Y 438.848,Z 462.868,A -85,B 0,C 180,E1 -9081.48,E2 -9081.48} C_VEL
LIN {X 0,Y 438.614,Z 467.822,A -85,B 0,C 180,E1 -9082.634,E2 -9082.634} C_VEL
LIN {X 0,Y 438.405,Z 472.46,A -85,B 0,C 180,E1 -9083.963,E2 -9083.963} C_VEL
LIN {X 0,Y 438.348,Z 476.312,A -85,B 0,C 180,E1 -9085.401,E2 -9085.401} C_VEL
LIN {X 0,Y 438.262,Z 478.213,A -85,B 0,C 180,E1 -9086.321,E2 -9086.321} C_VEL
LIN {X 0,Y 438.297,Z 479.664,A -85,B 0,C 180,E1 -9087.241,E2 -9087.241} C_VEL
LIN {X 0,Y 438.277,Z 480.688,A -85,B 0,C 180,E1 -9088.161,E2 -9088.161} C_VEL
LIN {X 0,Y 438.232,Z 481.571,A -85,B 0,C 180,E1 -9089.999,E2 -9089.999} C_VEL
LIN {X 0,Y 438.233,Z 481.402,A -85,B 0,C 180,E1 -9090.917,E2 -9090.917} C_VEL
LIN {X 0,Y 438.276,Z 480.821,A -85,B 0,C 180,E1 -9091.836,E2 -9091.836} C_VEL
LIN {X 0,Y 438.296,Z 479.852,A -85,B 0,C 180,E1 -9092.756,E2 -9092.756} C_VEL
LIN {X 0,Y 438.262,Z 478.488,A -85,B 0,C 180,E1 -9093.676,E2 -9093.676} C_VEL
LIN {X 0,Y 438.422,Z 475.607,A -85,B 0,C 180,E1 -9095.057,E2 -9095.057} C_VEL
LIN {X 0,Y 438.473,Z 471.698,A -85,B 0,C 180,E1 -9096.441,E2 -9096.441} C_VEL
LIN {X 0,Y 438.708,Z 466.662,A -85,B 0,C 180,E1 -9097.825,E2 -9097.825} C_VEL
LIN {X 0,Y 439.066,Z 460.339,A -85,B 0,C 180,E1 -9099.209,E2 -9099.209} C_VEL
LIN {X 0,Y 439.53,Z 452.44,A -85,B 0,C 180,E1 -9100.594,E2 -9100.594} C_VEL
LIN {X 0,Y 440.103,Z 444.403,A -85,B 0,C 180,E1 -9101.746,E2 -9101.746} C_VEL
LIN {X 0,Y 440.751,Z 434.611,A -85,B 0,C 180,E1 -9102.898,E2 -9102.898} C_VEL
LIN {X 0,Y 441.38,Z 423.691,A -85,B 0,C 180,E1 -9103.934,E2 -9103.934} C_VEL
LIN {X 0,Y 442.077,Z 411.243,A -85,B 0,C 180,E1 -9104.852,E2 -9104.852} C_VEL
LIN {X 0,Y 442.779,Z 399.015,A -85,B 0,C 180,E1 -9105.535,E2 -9105.535} C_VEL
LIN {X 0,Y 443.212,Z 386.141,A -85,B 0,C 180,E1 -9106.05,E2 -9106.05} C_VEL
LIN {X 0,Y 443.632,Z 372.495,A -85,B 0,C 180,E1 -9106.389,E2 -9106.389} C_VEL
LIN {X 0,Y 444.334,Z 290.251,A -85,B 0,C 180,E1 -9107.759,E2 -9107.759} C_VEL
LIN {X 0,Y 440.736,Z 269.645,A -85,B 0,C 180,E1 -9108.298,E2 -9108.298} C_VEL
LIN {X 0,Y 441.08,Z 261.812,A -85,B 0,C 180,E1 -9109.784,E2 -9109.784} C_VEL
LIN {X 0,Y 441.979,Z 245.729,A -85,B 0,C 180,E1 -9112.999,E2 -9112.999} C_VEL
LIN {X 0,Y 440.055,Z 235.252,A -85,B 0,C 180,E1 -9115.289,E2 -9115.289} C_VEL
LIN {X 0,Y 439.435,Z 232.317,A -85,B 0,C 180,E1 -9116.004,E2 -9116.004} C_VEL
LIN {X 0,Y 439.421,Z 232.247,A -85,B 0,C 180,E1 -9118.671,E2 -9118.671} C_VEL
LIN {X 0,Y 439.372,Z 232.254,A -85,B 0,C 180,E1 -9122.028,E2 -9122.028} C_VEL
LIN {X 0,Y 439.395,Z 232.246,A -85,B 0,C 180,E1 -9125.337,E2 -9125.337} C_VEL
LIN {X 0,Y 439.364,Z 232.252,A -85,B 0,C 180,E1 -9128.595,E2 -9128.595} C_VEL
LIN {X 0,Y 439.382,Z 232.249,A -85,B 0,C 180,E1 -9131.253,E2 -9131.253} C_VEL
LIN {X 0,Y 439.377,Z 232.252,A -85,B 0,C 180,E1 -9134.73,E2 -9134.73} C_VEL
LIN {X 0,Y 439.381,Z 232.245,A -85,B 0,C 180,E1 -9137.791,E2 -9137.791} C_VEL
LIN {X 0,Y 439.36,Z 232.252,A -85,B 0,C 180,E1 -9141.4,E2 -9141.4} C_VEL
LIN {X 0,Y 439.395,Z 232.253,A -85,B 0,C 180,E1 -9144.841,E2 -9144.841} C_VEL
LIN {X 0,Y 439.369,Z 232.251,A -85,B 0,C 180,E1 -9148.136,E2 -9148.136} C_VEL
LIN {X 0,Y 439.399,Z 232.246,A -85,B 0,C 180,E1 -9151.602,E2 -9151.602} C_VEL
LIN {X 0,Y 439.361,Z 232.254,A -85,B 0,C 180,E1 -9154.41,E2 -9154.41} C_VEL
LIN {X 0,Y 439.356,Z 232.253,A -85,B 0,C 180,E1 -9157.421,E2 -9157.421} C_VEL
LIN {X 0,Y 439.434,Z 232.245,A -85,B 0,C 180,E1 -9160.66,E2 -9160.66} C_VEL
LIN {X 0,Y 439.452,Z 232.238,A -85,B 0,C 180,E1 -9164.221,E2 -9164.221} C_VEL
LIN {X 0,Y 439.472,Z 232.234,A -85,B 0,C 180,E1 -9167.998,E2 -9167.998} C_VEL
LIN {X 0,Y 439.472,Z 232.235,A -85,B 0,C 180,E1 -9171.722,E2 -9171.722} C_VEL
LIN {X 0,Y 439.594,Z 232.223,A -85,B 0,C 180,E1 -9174.492,E2 -9174.492} C_VEL
LIN {X 0,Y 439.609,Z 232.222,A -85,B 0,C 180,E1 -9178.164,E2 -9178.164} C_VEL
LIN {X 0,Y 439.632,Z 232.218,A -85,B 0,C 180,E1 -9179.996,E2 -9179.996} C_VEL
LIN {X 0,Y 439.59,Z 232.223,A -85,B 0,C 180,E1 -9182.745,E2 -9182.745} C_VEL
LIN {X 0,Y 439.539,Z 232.23,A -85,B 0,C 180,E1 -9186.423,E2 -9186.423} C_VEL
LIN {X 0,Y 439.474,Z 232.238,A -85,B 0,C 180,E1 -9189.198,E2 -9189.198} C_VEL
LIN {X 0,Y 439.444,Z 232.239,A -85,B 0,C 180,E1 -9192.934,E2 -9192.934} C_VEL
LIN {X 0,Y 439.423,Z 232.245,A -85,B 0,C 180,E1 -9196.344,E2 -9196.344} C_VEL
LIN {X 0,Y 439.377,Z 232.253,A -85,B 0,C 180,E1 -9199.623,E2 -9199.623} C_VEL
LIN {X 0,Y 439.337,Z 232.258,A -85,B 0,C 180,E1 -9202.572,E2 -9202.572} C_VEL
LIN {X 0,Y 439.369,Z 232.25,A -85,B 0,C 180,E1 -9205.582,E2 -9205.582} C_VEL
LIN {X 0,Y 439.388,Z 232.245,A -85,B 0,C 180,E1 -9208.67,E2 -9208.67} C_VEL
LIN {X 0,Y 439.339,Z 232.257,A -85,B 0,C 180,E1 -9212.027,E2 -9212.027} C_VEL
LIN {X 0,Y 439.364,Z 232.25,A -85,B 0,C 180,E1 -9215.338,E2 -9215.338} C_VEL
LIN {X 0,Y 439.365,Z 232.255,A -85,B 0,C 180,E1 -9218.591,E2 -9218.591} C_VEL
LIN {X 0,Y 439.369,Z 232.257,A -85,B 0,C 180,E1 -9221.257,E2 -9221.257} C_VEL
LIN {X 0,Y 439.374,Z 232.256,A -85,B 0,C 180,E1 -9224.726,E2 -9224.726} C_VEL
LIN {X 0,Y 439.4,Z 232.436,A -85,B 0,C 180,E1 -9225.273,E2 -9225.273} C_VEL
LIN {X 0,Y 441.368,Z 242.56,A -85,B 0,C 180,E1 -9227.565,E2 -9227.565} C_VEL
LIN {X 0,Y 441.045,Z 252.452,A -85,B 0,C 180,E1 -9229.606,E2 -9229.606} C_VEL
LIN {X 0,Y 440.814,Z 258.181,A -85,B 0,C 180,E1 -9230.726,E2 -9230.726} C_VEL
LIN {X 0,Y 442.06,Z 264.173,A -85,B 0,C 180,E1 -9230.928,E2 -9230.928} C_VEL
LIN {X 0,Y 444.466,Z 276.913,A -85,B 0,C 180,E1 -9231.259,E2 -9231.259} C_VEL
LIN {X 0,Y 443.568,Z 365.684,A -85,B 0,C 180,E1 -9232.751,E2 -9232.751} C_VEL
LIN {X 0,Y 443.138,Z 378.979,A -85,B 0,C 180,E1 -9233.154,E2 -9233.154} C_VEL
LIN {X 0,Y 442.664,Z 391.922,A -85,B 0,C 180,E1 -9233.746,E2 -9233.746} C_VEL
LIN {X 0,Y 442.024,Z 404.365,A -85,B 0,C 180,E1 -9234.528,E2 -9234.528} C_VEL
LIN {X 0,Y 441.344,Z 415.454,A -85,B 0,C 180,E1 -9235.426,E2 -9235.426} C_VEL
LIN {X 0,Y 440.682,Z 425.897,A -85,B 0,C 180,E1 -9236.484,E2 -9236.484} C_VEL
LIN {X 0,Y 440.069,Z 435.651,A -85,B 0,C 180,E1 -9237.722,E2 -9237.722} C_VEL
LIN {X 0,Y 439.521,Z 443.607,A -85,B 0,C 180,E1 -9238.959,E2 -9238.959} C_VEL
LIN {X 0,Y 439.111,Z 450.424,A -85,B 0,C 180,E1 -9240.256,E2 -9240.256} C_VEL
LIN {X 0,Y 438.798,Z 456.695,A -85,B 0,C 180,E1 -9241.74,E2 -9241.74} C_VEL
LIN {X 0,Y 438.499,Z 461.852,A -85,B 0,C 180,E1 -9243.337,E2 -9243.337} C_VEL
LIN {X 0,Y 438.308,Z 465.443,A -85,B 0,C 180,E1 -9244.857,E2 -9244.857} C_VEL
LIN {X 0,Y 438.156,Z 467.838,A -85,B 0,C 180,E1 -9246.361,E2 -9246.361} C_VEL
LIN {X 0,Y 438.063,Z 469.069,A -85,B 0,C 180,E1 -9247.812,E2 -9247.812} C_VEL
LIN {X 0,Y 438.09,Z 469.383,A -85,B 0,C 180,E1 -9249.335,E2 -9249.335} C_VEL
LIN {X 0,Y 438.172,Z 468.332,A -85,B 0,C 180,E1 -9251.124,E2 -9251.124} C_VEL
LIN {X 0,Y 438.168,Z 467.458,A -85,B 0,C 180,E1 -9251.801,E2 -9251.801} C_VEL
LIN {X 0,Y 437.526,Z 466.385,A -85,B 0,C 180,E1 -9252.556,E2 -9252.556} C_VEL
LIN {X 0,Y 434.759,Z 464.003,A -85,B 0,C 180,E1 -9253.77,E2 -9253.77} C_VEL
LIN {X 0,Y 432.464,Z 461.655,A -85,B 0,C 180,E1 -9254.73,E2 -9254.73} C_VEL
LIN {X 0,Y 431.545,Z 459.526,A -85,B 0,C 180,E1 -9255.455,E2 -9255.455} C_VEL
LIN {X 0,Y 431.506,Z 458.707,A -85,B 0,C 180,E1 -9255.697,E2 -9255.697} C_VEL
LIN {X 0,Y 431.805,Z 452.678,A -85,B 0,C 180,E1 -9257.275,E2 -9257.275} C_VEL
LIN {X 0,Y 432.222,Z 445.486,A -85,B 0,C 180,E1 -9258.75,E2 -9258.75} C_VEL
LIN {X 0,Y 432.636,Z 438.29,A -85,B 0,C 180,E1 -9259.944,E2 -9259.944} C_VEL
LIN {X 0,Y 433.271,Z 428.46,A -85,B 0,C 180,E1 -9261.267,E2 -9261.267} C_VEL
LIN {X 0,Y 433.962,Z 417.576,A -85,B 0,C 180,E1 -9262.44,E2 -9262.44} C_VEL
LIN {X 0,Y 434.616,Z 406.493,A -85,B 0,C 180,E1 -9263.385,E2 -9263.385} C_VEL
LIN {X 0,Y 435.224,Z 394.069,A -85,B 0,C 180,E1 -9264.209,E2 -9264.209} C_VEL
LIN {X 0,Y 435.69,Z 382.3,A -85,B 0,C 180,E1 -9264.796,E2 -9264.796} C_VEL
LIN {X 0,Y 436.119,Z 369.552,A -85,B 0,C 180,E1 -9265.235,E2 -9265.235} C_VEL
LIN {X 0,Y 436.314,Z 352.679,A -85,B 0,C 180,E1 -9265.573,E2 -9265.573} C_VEL
LIN {X 0,Y 436.972,Z 277.323,A -85,B 0,C 180,E1 -9266.832,E2 -9266.832} C_VEL
LIN {X 0,Y 433.662,Z 258.745,A -85,B 0,C 180,E1 -9267.302,E2 -9267.302} C_VEL
LIN {X 0,Y 433.699,Z 256.603,A -85,B 0,C 180,E1 -9267.68,E2 -9267.68} C_VEL
LIN {X 0,Y 434.33,Z 244.727,A -85,B 0,C 180,E1 -9270.233,E2 -9270.233} C_VEL
LIN {X 0,Y 433.888,Z 240.597,A -85,B 0,C 180,E1 -9271.162,E2 -9271.162} C_VEL
LIN {X 0,Y 432.531,Z 233.226,A -85,B 0,C 180,E1 -9272.912,E2 -9272.912} C_VEL
LIN {X 0,Y 432.528,Z 233.107,A -85,B 0,C 180,E1 -9276.532,E2 -9276.532} C_VEL
LIN {X 0,Y 432.402,Z 233.124,A -85,B 0,C 180,E1 -9279.355,E2 -9279.355} C_VEL
LIN {X 0,Y 432.405,Z 233.118,A -85,B 0,C 180,E1 -9282.814,E2 -9282.814} C_VEL
LIN {X 0,Y 432.374,Z 233.122,A -85,B 0,C 180,E1 -9286.481,E2 -9286.481} C_VEL
LIN {X 0,Y 432.301,Z 233.138,A -85,B 0,C 180,E1 -9289.964,E2 -9289.964} C_VEL
LIN {X 0,Y 432.28,Z 233.133,A -85,B 0,C 180,E1 -9292.968,E2 -9292.968} C_VEL
LIN {X 0,Y 432.301,Z 233.131,A -85,B 0,C 180,E1 -9295.006,E2 -9295.006} C_VEL
LIN {X 0,Y 432.31,Z 233.138,A -85,B 0,C 180,E1 -9298.13,E2 -9298.13} C_VEL
LIN {X 0,Y 432.287,Z 233.132,A -85,B 0,C 180,E1 -9301.35,E2 -9301.35} C_VEL
LIN {X 0,Y 432.296,Z 233.135,A -85,B 0,C 180,E1 -9304.683,E2 -9304.683} C_VEL
LIN {X 0,Y 432.294,Z 233.136,A -85,B 0,C 180,E1 -9308.156,E2 -9308.156} C_VEL
LIN {X 0,Y 432.279,Z 233.134,A -85,B 0,C 180,E1 -9311.805,E2 -9311.805} C_VEL
LIN {X 0,Y 432.31,Z 233.133,A -85,B 0,C 180,E1 -9314.352,E2 -9314.352} C_VEL
LIN {X 0,Y 432.285,Z 233.137,A -85,B 0,C 180,E1 -9317.022,E2 -9317.022} C_VEL
LIN {X 0,Y 432.271,Z 233.134,A -85,B 0,C 180,E1 -9319.832,E2 -9319.832} C_VEL
LIN {X 0,Y 432.289,Z 233.14,A -85,B 0,C 180,E1 -9323.026,E2 -9323.026} C_VEL
LIN {X 0,Y 432.318,Z 233.128,A -85,B 0,C 180,E1 -9326.007,E2 -9326.007} C_VEL
LIN {X 0,Y 432.328,Z 233.131,A -85,B 0,C 180,E1 -9329.496,E2 -9329.496} C_VEL
LIN {X 0,Y 432.308,Z 233.131,A -85,B 0,C 180,E1 -9331.877,E2 -9331.877} C_VEL
LIN {X 0,Y 432.311,Z 233.133,A -85,B 0,C 180,E1 -9335.001,E2 -9335.001} C_VEL
LIN {X 0,Y 432.351,Z 233.126,A -85,B 0,C 180,E1 -9338.05,E2 -9338.05} C_VEL
LIN {X 0,Y 432.379,Z 233.123,A -85,B 0,C 180,E1 -9341.034,E2 -9341.034} C_VEL
LIN {X 0,Y 432.423,Z 233.119,A -85,B 0,C 180,E1 -9343.965,E2 -9343.965} C_VEL
LIN {X 0,Y 432.454,Z 233.119,A -85,B 0,C 180,E1 -9347.807,E2 -9347.807} C_VEL
LIN {X 0,Y 432.449,Z 233.117,A -85,B 0,C 180,E1 -9351.593,E2 -9351.593} C_VEL
LIN {X 0,Y 432.554,Z 233.102,A -85,B 0,C 180,E1 -9354.409,E2 -9354.409} C_VEL
LIN {X 0,Y 432.602,Z 233.101,A -85,B 0,C 180,E1 -9358.142,E2 -9358.142} C_VEL
LIN {X 0,Y 432.543,Z 233.101,A -85,B 0,C 180,E1 -9360.935,E2 -9360.935} C_VEL
LIN {X 0,Y 432.563,Z 233.1,A -85,B 0,C 180,E1 -9362.797,E2 -9362.797} C_VEL
LIN {X 0,Y 432.524,Z 233.109,A -85,B 0,C 180,E1 -9366.534,E2 -9366.534} C_VEL
LIN {X 0,Y 432.434,Z 233.114,A -85,B 0,C 180,E1 -9369.357,E2 -9369.357} C_VEL
LIN {X 0,Y 432.443,Z 233.118,A -85,B 0,C 180,E1 -9372.806,E2 -9372.806} C_VEL
LIN {X 0,Y 432.425,Z 233.121,A -85,B 0,C 180,E1 -9376.481,E2 -9376.481} C_VEL
LIN {X 0,Y 432.351,Z 233.124,A -85,B 0,C 180,E1 -9379.963,E2 -9379.963} C_VEL
LIN {X 0,Y 432.324,Z 233.135,A -85,B 0,C 180,E1 -9382.967,E2 -9382.967} C_VEL
LIN {X 0,Y 432.334,Z 233.127,A -85,B 0,C 180,E1 -9386.037,E2 -9386.037} C_VEL
LIN {X 0,Y 432.337,Z 233.133,A -85,B 0,C 180,E1 -9389.191,E2 -9389.191} C_VEL
LIN {X 0,Y 432.335,Z 233.127,A -85,B 0,C 180,E1 -9392.445,E2 -9392.445} C_VEL
LIN {X 0,Y 432.351,Z 233.127,A -85,B 0,C 180,E1 -9395.819,E2 -9395.819} C_VEL
LIN {X 0,Y 432.317,Z 233.136,A -85,B 0,C 180,E1 -9399.349,E2 -9399.349} C_VEL
LIN {X 0,Y 432.318,Z 233.133,A -85,B 0,C 180,E1 -9401.802,E2 -9401.802} C_VEL
LIN {X 0,Y 432.347,Z 233.125,A -85,B 0,C 180,E1 -9404.348,E2 -9404.348} C_VEL
LIN {X 0,Y 432.317,Z 233.13,A -85,B 0,C 180,E1 -9407.019,E2 -9407.019} C_VEL
LIN {X 0,Y 432.304,Z 233.138,A -85,B 0,C 180,E1 -9409.828,E2 -9409.828} C_VEL
LIN {X 0,Y 432.319,Z 233.129,A -85,B 0,C 180,E1 -9413.022,E2 -9413.022} C_VEL
LIN {X 0,Y 432.374,Z 233.13,A -85,B 0,C 180,E1 -9415.997,E2 -9415.997} C_VEL
LIN {X 0,Y 432.361,Z 233.124,A -85,B 0,C 180,E1 -9419.49,E2 -9419.49} C_VEL
LIN {X 0,Y 432.358,Z 233.13,A -85,B 0,C 180,E1 -9421.874,E2 -9421.874} C_VEL
LIN {X 0,Y 432.465,Z 233.345,A -85,B 0,C 180,E1 -9424.232,E2 -9424.232} C_VEL
LIN {X 0,Y 434.703,Z 245.728,A -85,B 0,C 180,E1 -9426.941,E2 -9426.941} C_VEL
LIN {X 0,Y 434.175,Z 256.552,A -85,B 0,C 180,E1 -9429.137,E2 -9429.137} C_VEL
LIN {X 0,Y 433.501,Z 269.491,A -85,B 0,C 180,E1 -9431.701,E2 -9431.701} C_VEL
LIN {X 0,Y 434.243,Z 274.488,A -85,B 0,C 180,E1 -9431.865,E2 -9431.865} C_VEL
LIN {X 0,Y 437.043,Z 291.913,A -85,B 0,C 180,E1 -9432.268,E2 -9432.268} C_VEL
LIN {X 0,Y 436.132,Z 377.58,A -85,B 0,C 180,E1 -9433.709,E2 -9433.709} C_VEL
LIN {X 0,Y 435.712,Z 390.766,A -85,B 0,C 180,E1 -9434.114,E2 -9434.114} C_VEL
LIN {X 0,Y 435.215,Z 402.905,A -85,B 0,C 180,E1 -9434.666,E2 -9434.666} C_VEL
LIN {X 0,Y 434.614,Z 414.35,A -85,B 0,C 180,E1 -9435.363,E2 -9435.363} C_VEL
LIN {X 0,Y 434.006,Z 425.603,A -85,B 0,C 180,E1 -9436.253,E2 -9436.253} C_VEL
LIN {X 0,Y 433.389,Z 436.669,A -85,B 0,C 180,E1 -9437.353,E2 -9437.353} C_VEL
LIN {X 0,Y 432.774,Z 446.169,A -85,B 0,C 180,E1 -9438.524,E2 -9438.524} C_VEL
LIN {X 0,Y 432.204,Z 455.306,A -85,B 0,C 180,E1 -9439.931,E2 -9439.931} C_VEL
LIN {X 0,Y 431.815,Z 462.663,A -85,B 0,C 180,E1 -9441.34,E2 -9441.34} C_VEL
LIN {X 0,Y 431.543,Z 467.642,A -85,B 0,C 180,E1 -9442.512,E2 -9442.512} C_VEL
LIN {X 0,Y 431.307,Z 472.729,A -85,B 0,C 180,E1 -9444.003,E2 -9444.003} C_VEL
LIN {X 0,Y 431.279,Z 476.172,A -85,B 0,C 180,E1 -9445.325,E2 -9445.325} C_VEL
LIN {X 0,Y 431.172,Z 478.08,A -85,B 0,C 180,E1 -9446.26,E2 -9446.26} C_VEL
LIN {X 0,Y 431.193,Z 479.544,A -85,B 0,C 180,E1 -9447.196,E2 -9447.196} C_VEL
LIN {X 0,Y 431.2,Z 480.574,A -85,B 0,C 180,E1 -9448.131,E2 -9448.131} C_VEL
LIN {X 0,Y 431.147,Z 481.47,A -85,B 0,C 180,E1 -9449.999,E2 -9449.999} C_VEL
LIN {X 0,Y 431.152,Z 481.313,A -85,B 0,C 180,E1 -9450.933,E2 -9450.933} C_VEL
LIN {X 0,Y 431.2,Z 480.738,A -85,B 0,C 180,E1 -9451.867,E2 -9451.867} C_VEL
LIN {X 0,Y 431.192,Z 479.775,A -85,B 0,C 180,E1 -9452.801,E2 -9452.801} C_VEL
LIN {X 0,Y 431.171,Z 478.42,A -85,B 0,C 180,E1 -9453.737,E2 -9453.737} C_VEL
LIN {X 0,Y 431.335,Z 475.556,A -85,B 0,C 180,E1 -9455.14,E2 -9455.14} C_VEL
LIN {X 0,Y 431.391,Z 471.669,A -85,B 0,C 180,E1 -9456.547,E2 -9456.547} C_VEL
LIN {X 0,Y 431.658,Z 466.661,A -85,B 0,C 180,E1 -9457.953,E2 -9457.953} C_VEL
LIN {X 0,Y 432.026,Z 460.376,A -85,B 0,C 180,E1 -9459.361,E2 -9459.361} C_VEL
LIN {X 0,Y 432.54,Z 452.514,A -85,B 0,C 180,E1 -9460.768,E2 -9460.768} C_VEL
LIN {X 0,Y 433.157,Z 444.511,A -85,B 0,C 180,E1 -9461.937,E2 -9461.937} C_VEL
LIN {X 0,Y 433.841,Z 434.759,A -85,B 0,C 180,E1 -9463.107,E2 -9463.107} C_VEL
LIN {X 0,Y 434.487,Z 423.914,A -85,B 0,C 180,E1 -9464.16,E2 -9464.16} C_VEL
LIN {X 0,Y 435.25,Z 411.55,A -85,B 0,C 180,E1 -9465.09,E2 -9465.09} C_VEL
LIN {X 0,Y 435.975,Z 399.439,A -85,B 0,C 180,E1 -9465.783,E2 -9465.783} C_VEL
LIN {X 0,Y 436.433,Z 386.883,A -85,B 0,C 180,E1 -9466.306,E2 -9466.306} C_VEL
LIN {X 0,Y 436.879,Z 373.775,A -85,B 0,C 180,E1 -9466.65,E2 -9466.65} C_VEL
LIN {X 0,Y 437.669,Z 291.278,A -85,B 0,C 180,E1 -9468.048,E2 -9468.048} C_VEL
LIN {X 0,Y 433.836,Z 269.514,A -85,B 0,C 180,E1 -9468.638,E2 -9468.638} C_VEL
LIN {X 0,Y 434.135,Z 263.068,A -85,B 0,C 180,E1 -9469.873,E2 -9469.873} C_VEL
LIN {X 0,Y 435.077,Z 247.849,A -85,B 0,C 180,E1 -9472.961,E2 -9472.961} C_VEL
LIN {X 0,Y 433.684,Z 239.337,A -85,B 0,C 180,E1 -9474.834,E2 -9474.834} C_VEL
LIN {X 0,Y 432.442,Z 233.399,A -85,B 0,C 180,E1 -9476.211,E2 -9476.211} C_VEL
LIN {X 0,Y 432.396,Z 233.127,A -85,B 0,C 180,E1 -9476.623,E2 -9476.623} C_VEL
LIN {X 0,Y 432.346,Z 233.129,A -85,B 0,C 180,E1 -9479.185,E2 -9479.185} C_VEL
LIN {X 0,Y 432.326,Z 233.129,A -85,B 0,C 180,E1 -9482.441,E2 -9482.441} C_VEL
LIN {X 0,Y 432.345,Z 233.126,A -85,B 0,C 180,E1 -9485.629,E2 -9485.629} C_VEL
LIN {X 0,Y 432.328,Z 233.129,A -85,B 0,C 180,E1 -9488.709,E2 -9488.709} C_VEL
LIN {X 0,Y 432.325,Z 233.127,A -85,B 0,C 180,E1 -9491.796,E2 -9491.796} C_VEL
LIN {X 0,Y 432.333,Z 233.134,A -85,B 0,C 180,E1 -9494.345,E2 -9494.345} C_VEL
LIN {X 0,Y 432.316,Z 233.124,A -85,B 0,C 180,E1 -9497.014,E2 -9497.014} C_VEL
LIN {X 0,Y 432.29,Z 233.136,A -85,B 0,C 180,E1 -9499.825,E2 -9499.825} C_VEL
LIN {X 0,Y 432.302,Z 233.132,A -85,B 0,C 180,E1 -9503.019,E2 -9503.019} C_VEL
LIN {X 0,Y 432.357,Z 233.127,A -85,B 0,C 180,E1 -9505.994,E2 -9505.994} C_VEL
LIN {X 0,Y 432.343,Z 233.127,A -85,B 0,C 180,E1 -9509.487,E2 -9509.487} C_VEL
LIN {X 0,Y 432.338,Z 233.126,A -85,B 0,C 180,E1 -9511.871,E2 -9511.871} C_VEL
LIN {X 0,Y 432.318,Z 233.131,A -85,B 0,C 180,E1 -9514.994,E2 -9514.994} C_VEL
LIN {X 0,Y 432.35,Z 233.124,A -85,B 0,C 180,E1 -9518.042,E2 -9518.042} C_VEL
LIN {X 0,Y 432.377,Z 233.129,A -85,B 0,C 180,E1 -9521.026,E2 -9521.026} C_VEL
LIN {X 0,Y 432.421,Z 233.114,A -85,B 0,C 180,E1 -9523.958,E2 -9523.958} C_VEL
LIN {X 0,Y 432.449,Z 233.11,A -85,B 0,C 180,E1 -9527.8,E2 -9527.8} C_VEL
LIN {X 0,Y 432.438,Z 233.112,A -85,B 0,C 180,E1 -9531.586,E2 -9531.586} C_VEL
LIN {X 0,Y 432.57,Z 233.098,A -85,B 0,C 180,E1 -9534.402,E2 -9534.402} C_VEL
LIN {X 0,Y 432.579,Z 233.098,A -85,B 0,C 180,E1 -9538.134,E2 -9538.134} C_VEL
LIN {X 0,Y 432.584,Z 233.096,A -85,B 0,C 180,E1 -9539.996,E2 -9539.996} C_VEL
LIN {X 0,Y 432.544,Z 233.101,A -85,B 0,C 180,E1 -9542.79,E2 -9542.79} C_VEL
LIN {X 0,Y 432.496,Z 233.107,A -85,B 0,C 180,E1 -9546.528,E2 -9546.528} C_VEL
LIN {X 0,Y 432.418,Z 233.118,A -85,B 0,C 180,E1 -9549.35,E2 -9549.35} C_VEL
LIN {X 0,Y 432.41,Z 233.115,A -85,B 0,C 180,E1 -9552.8,E2 -9552.8} C_VEL
LIN {X 0,Y 432.389,Z 233.121,A -85,B 0,C 180,E1 -9556.475,E2 -9556.475} C_VEL
LIN {X 0,Y 432.313,Z 233.133,A -85,B 0,C 180,E1 -9559.957,E2 -9559.957} C_VEL
LIN {X 0,Y 432.291,Z 233.133,A -85,B 0,C 180,E1 -9562.961,E2 -9562.961} C_VEL
LIN {X 0,Y 432.333,Z 233.131,A -85,B 0,C 180,E1 -9566.029,E2 -9566.029} C_VEL
LIN {X 0,Y 432.313,Z 233.127,A -85,B 0,C 180,E1 -9569.184,E2 -9569.184} C_VEL
LIN {X 0,Y 432.292,Z 233.132,A -85,B 0,C 180,E1 -9572.44,E2 -9572.44} C_VEL
LIN {X 0,Y 432.313,Z 233.128,A -85,B 0,C 180,E1 -9575.629,E2 -9575.629} C_VEL
LIN {X 0,Y 432.326,Z 233.132,A -85,B 0,C 180,E1 -9578.715,E2 -9578.715} C_VEL
LIN {X 0,Y 432.338,Z 233.131,A -85,B 0,C 180,E1 -9581.79,E2 -9581.79} C_VEL
LIN {X 0,Y 432.365,Z 233.301,A -85,B 0,C 180,E1 -9584.991,E2 -9584.991} C_VEL
LIN {X 0,Y 434.492,Z 244.31,A -85,B 0,C 180,E1 -9587.527,E2 -9587.527} C_VEL
LIN {X 0,Y 433.918,Z 257.609,A -85,B 0,C 180,E1 -9590.287,E2 -9590.287} C_VEL
LIN {X 0,Y 434.01,Z 258.89,A -85,B 0,C 180,E1 -9590.433,E2 -9590.433} C_VEL
LIN {X 0,Y 437.703,Z 277.579,A -85,B 0,C 180,E1 -9590.955,E2 -9590.955} C_VEL
LIN {X 0,Y 436.814,Z 366.238,A -85,B 0,C 180,E1 -9592.476,E2 -9592.476} C_VEL
LIN {X 0,Y 436.364,Z 379.799,A -85,B 0,C 180,E1 -9592.902,E2 -9592.902} C_VEL
LIN {X 0,Y 435.849,Z 392.603,A -85,B 0,C 180,E1 -9593.505,E2 -9593.505} C_VEL
LIN {X 0,Y 435.229,Z 403.967,A -85,B 0,C 180,E1 -9594.231,E2 -9594.231} C_VEL
LIN {X 0,Y 434.539,Z 414.713,A -85,B 0,C 180,E1 -9595.103,E2 -9595.103} C_VEL
LIN {X 0,Y 433.855,Z 425.194,A -85,B 0,C 180,E1 -9596.165,E2 -9596.165} C_VEL
LIN {X 0,Y 433.214,Z 434.705,A -85,B 0,C 180,E1 -9597.359,E2 -9597.359} C_VEL
LIN {X 0,Y 432.565,Z 443.187,A -85,B 0,C 180,E1 -9598.676,E2 -9598.676} C_VEL
LIN {X 0,Y 432.038,Z 451.342,A -85,B 0,C 180,E1 -9600.257,E2 -9600.257} C_VEL
LIN {X 0,Y 431.676,Z 457.623,A -85,B 0,C 180,E1 -9601.829,E2 -9601.829} C_VEL
LIN {X 0,Y 431.429,Z 462.145,A -85,B 0,C 180,E1 -9603.291,E2 -9603.291} C_VEL
LIN {X 0,Y 431.209,Z 465.857,A -85,B 0,C 180,E1 -9604.93,E2 -9604.93} C_VEL
LIN {X 0,Y 431.124,Z 467.521,A -85,B 0,C 180,E1 -9605.951,E2 -9605.951} C_VEL
LIN {X 0,Y 431.001,Z 468.64,A -85,B 0,C 180,E1 -9606.963,E2 -9606.963} C_VEL
LIN {X 0,Y 430.988,Z 469.448,A -85,B 0,C 180,E1 -9608.339,E2 -9608.339} C_VEL
LIN {X 0,Y 430.994,Z 469.27,A -85,B 0,C 180,E1 -9609.976,E2 -9609.976} C_VEL
LIN {X 0,Y 431.059,Z 468.548,A -85,B 0,C 180,E1 -9611.003,E2 -9611.003} C_VEL
LIN {X 0,Y 431.081,Z 467.453,A -85,B 0,C 180,E1 -9611.957,E2 -9611.957} C_VEL
LIN {X 0,Y 431.197,Z 464.886,A -85,B 0,C 180,E1 -9613.429,E2 -9613.429} C_VEL
LIN {X 0,Y 431.419,Z 461.24,A -85,B 0,C 180,E1 -9614.893,E2 -9614.893} C_VEL
LIN {X 0,Y 431.506,Z 458.707,A -85,B 0,C 180,E1 -9615.697,E2 -9615.697} C_VEL
LIN {X 0,Y 430.98,Z 456.256,A -85,B 0,C 180,E1 -9616.407,E2 -9616.407} C_VEL
LIN {X 0,Y 428.376,Z 451.826,A -85,B 0,C 180,E1 -9617.539,E2 -9617.539} C_VEL
LIN {X 0,Y 425.791,Z 446.795,A -85,B 0,C 180,E1 -9618.636,E2 -9618.636} C_VEL
LIN {X 0,Y 425.303,Z 443.331,A -85,B 0,C 180,E1 -9619.282,E2 -9619.282} C_VEL
LIN {X 0,Y 425.827,Z 435.617,A -85,B 0,C 180,E1 -9620.502,E2 -9620.502} C_VEL
LIN {X 0,Y 426.436,Z 426.773,A -85,B 0,C 180,E1 -9621.655,E2 -9621.655} C_VEL
LIN {X 0,Y 427.05,Z 417.235,A -85,B 0,C 180,E1 -9622.674,E2 -9622.674} C_VEL
LIN {X 0,Y 427.733,Z 406.01,A -85,B 0,C 180,E1 -9623.634,E2 -9623.634} C_VEL
LIN {X 0,Y 428.391,Z 393.422,A -85,B 0,C 180,E1 -9624.471,E2 -9624.471} C_VEL
LIN {X 0,Y 428.869,Z 380.642,A -85,B 0,C 180,E1 -9625.096,E2 -9625.096} C_VEL
LIN {X 0,Y 429.302,Z 366.884,A -85,B 0,C 180,E1 -9625.542,E2 -9625.542} C_VEL
LIN {X 0,Y 429.857,Z 314.745,A -85,B 0,C 180,E1 -9626.457,E2 -9626.457} C_VEL
LIN {X 0,Y 430.173,Z 278.472,A -85,B 0,C 180,E1 -9627.075,E2 -9627.075} C_VEL
LIN {X 0,Y 426.714,Z 258.914,A -85,B 0,C 180,E1 -9627.568,E2 -9627.568} C_VEL
LIN {X 0,Y 426.734,Z 257.152,A -85,B 0,C 180,E1 -9627.854,E2 -9627.854} C_VEL
LIN {X 0,Y 427.353,Z 245.167,A -85,B 0,C 180,E1 -9630.473,E2 -9630.473} C_VEL
LIN {X 0,Y 425.688,Z 235.026,A -85,B 0,C 180,E1 -9632.84,E2 -9632.84} C_VEL
LIN {X 0,Y 425.41,Z 234.009,A -85,B 0,C 180,E1 -9633.198,E2 -9633.198} C_VEL
LIN {X 0,Y 425.486,Z 233.984,A -85,B 0,C 180,E1 -9636.641,E2 -9636.641} C_VEL
LIN {X 0,Y 425.361,Z 234.003,A -85,B 0,C 180,E1 -9639.512,E2 -9639.512} C_VEL
LIN {X 0,Y 425.364,Z 233.995,A -85,B 0,C 180,E1 -9642.912,E2 -9642.912} C_VEL
LIN {X 0,Y 425.323,Z 234,A -85,B 0,C 180,E1 -9646.608,E2 -9646.608} C_VEL
LIN {X 0,Y 425.291,Z 234.009,A -85,B 0,C 180,E1 -9649.639,E2 -9649.639} C_VEL
LIN {X 0,Y 425.252,Z 234.012,A -85,B 0,C 180,E1 -9652.342,E2 -9652.342} C_VEL
LIN {X 0,Y 425.283,Z 234.006,A -85,B 0,C 180,E1 -9654.66,E2 -9654.66} C_VEL
LIN {X 0,Y 425.235,Z 234.012,A -85,B 0,C 180,E1 -9657.567,E2 -9657.567} C_VEL
LIN {X 0,Y 425.259,Z 234.01,A -85,B 0,C 180,E1 -9660.765,E2 -9660.765} C_VEL
LIN {X 0,Y 425.26,Z 234.015,A -85,B 0,C 180,E1 -9664.288,E2 -9664.288} C_VEL
LIN {X 0,Y 425.242,Z 234.01,A -85,B 0,C 180,E1 -9667.7,E2 -9667.7} C_VEL
LIN {X 0,Y 425.217,Z 234.021,A -85,B 0,C 180,E1 -9670.519,E2 -9670.519} C_VEL
LIN {X 0,Y 425.223,Z 234.013,A -85,B 0,C 180,E1 -9673.354,E2 -9673.354} C_VEL
LIN {X 0,Y 425.235,Z 234.012,A -85,B 0,C 180,E1 -9676.048,E2 -9676.048} C_VEL
LIN {X 0,Y 425.231,Z 234.017,A -85,B 0,C 180,E1 -9678.623,E2 -9678.623} C_VEL
LIN {X 0,Y 425.262,Z 234.013,A -85,B 0,C 180,E1 -9681.104,E2 -9681.104} C_VEL
LIN {X 0,Y 425.28,Z 234.009,A -85,B 0,C 180,E1 -9684.668,E2 -9684.668} C_VEL
LIN {X 0,Y 425.247,Z 234.009,A -85,B 0,C 180,E1 -9688.077,E2 -9688.077} C_VEL
LIN {X 0,Y 425.285,Z 234.011,A -85,B 0,C 180,E1 -9691.37,E2 -9691.37} C_VEL
LIN {X 0,Y 425.248,Z 234.01,A -85,B 0,C 180,E1 -9694.557,E2 -9694.557} C_VEL
LIN {X 0,Y 425.285,Z 234.009,A -85,B 0,C 180,E1 -9697.734,E2 -9697.734} C_VEL
LIN {X 0,Y 425.357,Z 233.996,A -85,B 0,C 180,E1 -9700.708,E2 -9700.708} C_VEL
LIN {X 0,Y 425.383,Z 234,A -85,B 0,C 180,E1 -9703.693,E2 -9703.693} C_VEL
LIN {X 0,Y 425.409,Z 233.995,A -85,B 0,C 180,E1 -9707.602,E2 -9707.602} C_VEL
LIN {X 0,Y 425.397,Z 233.993,A -85,B 0,C 180,E1 -9711.453,E2 -9711.453} C_VEL
LIN {X 0,Y 425.512,Z 233.98,A -85,B 0,C 180,E1 -9714.317,E2 -9714.317} C_VEL
LIN {X 0,Y 425.571,Z 233.977,A -85,B 0,C 180,E1 -9718.111,E2 -9718.111} C_VEL
LIN {X 0,Y 425.507,Z 233.977,A -85,B 0,C 180,E1 -9720.95,E2 -9720.95} C_VEL
LIN {X 0,Y 425.518,Z 233.977,A -85,B 0,C 180,E1 -9722.844,E2 -9722.844} C_VEL
LIN {X 0,Y 425.518,Z 233.977,A -85,B 0,C 180,E1 -9725.691,E2 -9725.691} C_VEL
LIN {X 0,Y 425.406,Z 233.996,A -85,B 0,C 180,E1 -9728.554,E2 -9728.554} C_VEL
LIN {X 0,Y 425.424,Z 233.993,A -85,B 0,C 180,E1 -9732.405,E2 -9732.405} C_VEL
LIN {X 0,Y 425.401,Z 233.994,A -85,B 0,C 180,E1 -9736.314,E2 -9736.314} C_VEL
LIN {X 0,Y 425.342,Z 233.998,A -85,B 0,C 180,E1 -9739.638,E2 -9739.638} C_VEL
LIN {X 0,Y 425.301,Z 234.004,A -85,B 0,C 180,E1 -9742.341,E2 -9742.341} C_VEL
LIN {X 0,Y 425.276,Z 234.008,A -85,B 0,C 180,E1 -9745.45,E2 -9745.45} C_VEL
LIN {X 0,Y 425.315,Z 234.006,A -85,B 0,C 180,E1 -9748.86,E2 -9748.86} C_VEL
LIN {X 0,Y 425.275,Z 234.006,A -85,B 0,C 180,E1 -9751.929,E2 -9751.929} C_VEL
LIN {X 0,Y 425.31,Z 234.01,A -85,B 0,C 180,E1 -9755.338,E2 -9755.338} C_VEL
LIN {X 0,Y 425.296,Z 234.005,A -85,B 0,C 180,E1 -9758.902,E2 -9758.902} C_VEL
LIN {X 0,Y 425.272,Z 234.006,A -85,B 0,C 180,E1 -9762.656,E2 -9762.656} C_VEL
LIN {X 0,Y 425.299,Z 234.007,A -85,B 0,C 180,E1 -9765.284,E2 -9765.284} C_VEL
LIN {X 0,Y 425.262,Z 234.008,A -85,B 0,C 180,E1 -9768.618,E2 -9768.618} C_VEL
LIN {X 0,Y 425.295,Z 234.004,A -85,B 0,C 180,E1 -9771.1,E2 -9771.1} C_VEL
LIN {X 0,Y 425.313,Z 234.002,A -85,B 0,C 180,E1 -9774.664,E2 -9774.664} C_VEL
LIN {X 0,Y 425.28,Z 234.014,A -85,B 0,C 180,E1 -9778.073,E2 -9778.073} C_VEL
LIN {X 0,Y 425.325,Z 234.005,A -85,B 0,C 180,E1 -9781.366,E2 -9781.366} C_VEL
LIN {X 0,Y 425.385,Z 234.096,A -85,B 0,C 180,E1 -9783.968,E2 -9783.968} C_VEL
LIN {X 0,Y 427.686,Z 246.521,A -85,B 0,C 180,E1 -9786.771,E2 -9786.771} C_VEL
LIN {X 0,Y 427.433,Z 253.862,A -85,B 0,C 180,E1 -9788.286,E2 -9788.286} C_VEL
LIN {X 0,Y 426.538,Z 269.358,A -85,B 0,C 180,E1 -9791.419,E2 -9791.419} C_VEL
LIN {X 0,Y 427.021,Z 272.865,A -85,B 0,C 180,E1 -9791.55,E2 -9791.55} C_VEL
LIN {X 0,Y 430.211,Z 292.5,A -85,B 0,C 180,E1 -9792.016,E2 -9792.016} C_VEL
LIN {X 0,Y 429.273,Z 377.432,A -85,B 0,C 180,E1 -9793.472,E2 -9793.472} C_VEL
LIN {X 0,Y 428.811,Z 390.629,A -85,B 0,C 180,E1 -9793.882,E2 -9793.882} C_VEL
LIN {X 0,Y 428.287,Z 403.345,A -85,B 0,C 180,E1 -9794.472,E2 -9794.472} C_VEL
LIN {X 0,Y 427.633,Z 415.437,A -85,B 0,C 180,E1 -9795.241,E2 -9795.241} C_VEL
LIN {X 0,Y 426.954,Z 427.276,A -85,B 0,C 180,E1 -9796.218,E2 -9796.218} C_VEL
LIN {X 0,Y 426.362,Z 437.365,A -85,B 0,C 180,E1 -9797.262,E2 -9797.262} C_VEL
LIN {X 0,Y 425.795,Z 445.848,A -85,B 0,C 180,E1 -9798.333,E2 -9798.333} C_VEL
LIN {X 0,Y 425.159,Z 455.029,A -85,B 0,C 180,E1 -9799.763,E2 -9799.763} C_VEL
LIN {X 0,Y 424.761,Z 462.419,A -85,B 0,C 180,E1 -9801.195,E2 -9801.195} C_VEL
LIN {X 0,Y 424.372,Z 469.191,A -85,B 0,C 180,E1 -9802.864,E2 -9802.864} C_VEL
LIN {X 0,Y 424.216,Z 473.653,A -85,B 0,C 180,E1 -9804.294,E2 -9804.294} C_VEL
LIN {X 0,Y 424.21,Z 476.007,A -85,B 0,C 180,E1 -9805.247,E2 -9805.247} C_VEL
LIN {X 0,Y 424.086,Z 477.926,A -85,B 0,C 180,E1 -9806.198,E2 -9806.198} C_VEL
LIN {X 0,Y 424.09,Z 479.411,A -85,B 0,C 180,E1 -9807.149,E2 -9807.149} C_VEL
LIN {X 0,Y 424.125,Z 480.452,A -85,B 0,C 180,E1 -9808.099,E2 -9808.099} C_VEL
LIN {X 0,Y 424.066,Z 481.366,A -85,B 0,C 180,E1 -9809.999,E2 -9809.999} C_VEL
LIN {X 0,Y 424.073,Z 481.228,A -85,B 0,C 180,E1 -9810.948,E2 -9810.948} C_VEL
LIN {X 0,Y 424.125,Z 480.664,A -85,B 0,C 180,E1 -9811.898,E2 -9811.898} C_VEL
LIN {X 0,Y 424.085,Z 478.365,A -85,B 0,C 180,E1 -9813.799,E2 -9813.799} C_VEL
LIN {X 0,Y 424.248,Z 475.521,A -85,B 0,C 180,E1 -9815.226,E2 -9815.226} C_VEL
LIN {X 0,Y 424.314,Z 471.655,A -85,B 0,C 180,E1 -9816.656,E2 -9816.656} C_VEL
LIN {X 0,Y 424.594,Z 466.668,A -85,B 0,C 180,E1 -9818.086,E2 -9818.086} C_VEL
LIN {X 0,Y 425.013,Z 460.41,A -85,B 0,C 180,E1 -9819.517,E2 -9819.517} C_VEL
LIN {X 0,Y 425.544,Z 452.588,A -85,B 0,C 180,E1 -9820.947,E2 -9820.947} C_VEL
LIN {X 0,Y 426.211,Z 444.618,A -85,B 0,C 180,E1 -9822.135,E2 -9822.135} C_VEL
LIN {X 0,Y 426.934,Z 434.907,A -85,B 0,C 180,E1 -9823.323,E2 -9823.323} C_VEL
LIN {X 0,Y 427.62,Z 424.125,A -85,B 0,C 180,E1 -9824.392,E2 -9824.392} C_VEL
LIN {X 0,Y 428.29,Z 413.618,A -85,B 0,C 180,E1 -9825.22,E2 -9825.22} C_VEL
LIN {X 0,Y 429.07,Z 400.986,A -85,B 0,C 180,E1 -9825.983,E2 -9825.983} C_VEL
LIN {X 0,Y 429.621,Z 388.394,A -85,B 0,C 180,E1 -9826.542,E2 -9826.542} C_VEL
LIN {X 0,Y 430.079,Z 376.511,A -85,B 0,C 180,E1 -9826.89,E2 -9826.89} C_VEL
LIN {X 0,Y 431.013,Z 292.386,A -85,B 0,C 180,E1 -9828.346,E2 -9828.346} C_VEL
LIN {X 0,Y 427.318,Z 271.56,A -85,B 0,C 180,E1 -9828.903,E2 -9828.903} C_VEL
LIN {X 0,Y 426.935,Z 269.174,A -85,B 0,C 180,E1 -9829.015,E2 -9829.015} C_VEL
LIN {X 0,Y 427.987,Z 252.285,A -85,B 0,C 180,E1 -9832.443,E2 -9832.443} C_VEL
LIN {X 0,Y 428.025,Z 247.458,A -85,B 0,C 180,E1 -9833.462,E2 -9833.462} C_VEL
LIN {X 0,Y 425.653,Z 235.482,A -85,B 0,C 180,E1 -9836.209,E2 -9836.209} C_VEL
LIN {X 0,Y 425.375,Z 234.022,A -85,B 0,C 180,E1 -9836.649,E2 -9836.649} C_VEL
LIN {X 0,Y 425.294,Z 234.013,A -85,B 0,C 180,E1 -9839.717,E2 -9839.717} C_VEL
LIN {X 0,Y 425.285,Z 234.005,A -85,B 0,C 180,E1 -9843.046,E2 -9843.046} C_VEL
LIN {X 0,Y 425.283,Z 234.008,A -85,B 0,C 180,E1 -9845.926,E2 -9845.926} C_VEL
LIN {X 0,Y 425.274,Z 234.007,A -85,B 0,C 180,E1 -9849.036,E2 -9849.036} C_VEL
LIN {X 0,Y 425.271,Z 234.006,A -85,B 0,C 180,E1 -9852.651,E2 -9852.651} C_VEL
LIN {X 0,Y 425.26,Z 234.005,A -85,B 0,C 180,E1 -9856.041,E2 -9856.041} C_VEL
LIN {X 0,Y 425.256,Z 234.015,A -85,B 0,C 180,E1 -9858.616,E2 -9858.616} C_VEL
LIN {X 0,Y 425.279,Z 234.007,A -85,B 0,C 180,E1 -9861.096,E2 -9861.096} C_VEL
LIN {X 0,Y 425.296,Z 234.009,A -85,B 0,C 180,E1 -9864.661,E2 -9864.661} C_VEL
LIN {X 0,Y 425.261,Z 234.008,A -85,B 0,C 180,E1 -9868.07,E2 -9868.07} C_VEL
LIN {X 0,Y 425.306,Z 234.003,A -85,B 0,C 180,E1 -9871.363,E2 -9871.363} C_VEL
LIN {X 0,Y 425.255,Z 234.011,A -85,B 0,C 180,E1 -9874.549,E2 -9874.549} C_VEL
LIN {X 0,Y 425.286,Z 234.005,A -85,B 0,C 180,E1 -9877.727,E2 -9877.727} C_VEL
LIN {X 0,Y 425.354,Z 234,A -85,B 0,C 180,E1 -9880.701,E2 -9880.701} C_VEL
LIN {X 0,Y 425.379,Z 233.992,A -85,B 0,C 180,E1 -9883.685,E2 -9883.685} C_VEL
LIN {X 0,Y 425.402,Z 233.988,A -85,B 0,C 180,E1 -9887.595,E2 -9887.595} C_VEL
LIN {X 0,Y 425.386,Z 233.992,A -85,B 0,C 180,E1 -9891.445,E2 -9891.445} C_VEL
LIN {X 0,Y 425.527,Z 233.976,A -85,B 0,C 180,E1 -9894.309,E2 -9894.309} C_VEL
LIN {X 0,Y 425.548,Z 233.974,A -85,B 0,C 180,E1 -9898.104,E2 -9898.104} C_VEL
LIN {X 0,Y 425.419,Z 233.988,A -85,B 0,C 180,E1 -9900.943,E2 -9900.943} C_VEL
LIN {X 0,Y 425.499,Z 233.979,A -85,B 0,C 180,E1 -9902.836,E2 -9902.836} C_VEL
LIN {X 0,Y 425.457,Z 233.984,A -85,B 0,C 180,E1 -9906.636,E2 -9906.636} C_VEL
LIN {X 0,Y 425.377,Z 233.995,A -85,B 0,C 180,E1 -9909.506,E2 -9909.506} C_VEL
LIN {X 0,Y 425.373,Z 233.992,A -85,B 0,C 180,E1 -9912.9,E2 -9912.9} C_VEL
LIN {X 0,Y 425.338,Z 233.998,A -85,B 0,C 180,E1 -9916.601,E2 -9916.601} C_VEL
LIN {X 0,Y 425.303,Z 234.006,A -85,B 0,C 180,E1 -9919.632,E2 -9919.632} C_VEL
LIN {X 0,Y 425.262,Z 234.011,A -85,B 0,C 180,E1 -9922.335,E2 -9922.335} C_VEL
LIN {X 0,Y 425.263,Z 234.007,A -85,B 0,C 180,E1 -9925.442,E2 -9925.442} C_VEL
LIN {X 0,Y 425.32,Z 234.002,A -85,B 0,C 180,E1 -9927.554,E2 -9927.554} C_VEL
LIN {X 0,Y 425.257,Z 234.013,A -85,B 0,C 180,E1 -9930.813,E2 -9930.813} C_VEL
LIN {X 0,Y 425.28,Z 234.012,A -85,B 0,C 180,E1 -9934.285,E2 -9934.285} C_VEL
LIN {X 0,Y 425.255,Z 234.012,A -85,B 0,C 180,E1 -9937.69,E2 -9937.69} C_VEL
LIN {X 0,Y 425.267,Z 234.011,A -85,B 0,C 180,E1 -9940.521,E2 -9940.521} C_VEL
LIN {X 0,Y 425.28,Z 234.011,A -85,B 0,C 180,E1 -9943.357,E2 -9943.357} C_VEL
LIN {X 0,Y 425.319,Z 234.082,A -85,B 0,C 180,E1 -9944.64,E2 -9944.64} C_VEL
LIN {X 0,Y 427.3,Z 244.025,A -85,B 0,C 180,E1 -9947.018,E2 -9947.018} C_VEL
LIN {X 0,Y 427.575,Z 248.358,A -85,B 0,C 180,E1 -9947.975,E2 -9947.975} C_VEL
LIN {X 0,Y 427.053,Z 258.321,A -85,B 0,C 180,E1 -9950.036,E2 -9950.036} C_VEL
LIN {X 0,Y 427.848,Z 262.225,A -85,B 0,C 180,E1 -9950.195,E2 -9950.195} C_VEL
LIN {X 0,Y 431.155,Z 279.15,A -85,B 0,C 180,E1 -9950.666,E2 -9950.666} C_VEL
LIN {X 0,Y 430.095,Z 366.127,A -85,B 0,C 180,E1 -9952.175,E2 -9952.175} C_VEL
LIN {X 0,Y 429.612,Z 379.73,A -85,B 0,C 180,E1 -9952.606,E2 -9952.606} C_VEL
LIN {X 0,Y 429.076,Z 392.52,A -85,B 0,C 180,E1 -9953.215,E2 -9953.215} C_VEL
LIN {X 0,Y 428.435,Z 403.943,A -85,B 0,C 180,E1 -9953.952,E2 -9953.952} C_VEL
LIN {X 0,Y 427.648,Z 415.277,A -85,B 0,C 180,E1 -9954.889,E2 -9954.889} C_VEL
LIN {X 0,Y 426.946,Z 425.684,A -85,B 0,C 180,E1 -9955.969,E2 -9955.969} C_VEL
LIN {X 0,Y 426.225,Z 435.427,A -85,B 0,C 180,E1 -9957.229,E2 -9957.229} C_VEL
LIN {X 0,Y 425.524,Z 444.289,A -85,B 0,C 180,E1 -9958.653,E2 -9958.653} C_VEL
LIN {X 0,Y 425.035,Z 451.057,A -85,B 0,C 180,E1 -9959.999,E2 -9959.999} C_VEL
LIN {X 0,Y 424.721,Z 456.463,A -85,B 0,C 180,E1 -9961.325,E2 -9961.325} C_VEL
LIN {X 0,Y 424.416,Z 461.582,A -85,B 0,C 180,E1 -9962.913,E2 -9962.913} C_VEL
LIN {X 0,Y 424.172,Z 465.306,A -85,B 0,C 180,E1 -9964.484,E2 -9964.484} C_VEL
LIN {X 0,Y 424.036,Z 467.386,A -85,B 0,C 180,E1 -9965.71,E2 -9965.71} C_VEL
LIN {X 0,Y 423.958,Z 468.433,A -85,B 0,C 180,E1 -9966.558,E2 -9966.558} C_VEL
LIN {X 0,Y 423.897,Z 469.526,A -85,B 0,C 180,E1 -9968.179,E2 -9968.179} C_VEL
LIN {X 0,Y 423.894,Z 469.523,A -85,B 0,C 180,E1 -9969.626,E2 -9969.626} C_VEL
LIN {X 0,Y 423.958,Z 468.759,A -85,B 0,C 180,E1 -9970.873,E2 -9970.873} C_VEL
LIN {X 0,Y 424.033,Z 466.532,A -85,B 0,C 180,E1 -9972.644,E2 -9972.644} C_VEL
LIN {X 0,Y 424.191,Z 463.998,A -85,B 0,C 180,E1 -9973.913,E2 -9973.913} C_VEL
LIN {X 0,Y 424.417,Z 458.967,A -85,B 0,C 180,E1 -9975.735,E2 -9975.735} C_VEL
LIN {X 0,Y 424.758,Z 452.487,A -85,B 0,C 180,E1 -9977.449,E2 -9977.449} C_VEL
LIN {X 0,Y 425.163,Z 445.991,A -85,B 0,C 180,E1 -9978.802,E2 -9978.802} C_VEL
LIN {X 0,Y 425.303,Z 443.331,A -85,B 0,C 180,E1 -9979.282,E2 -9979.282} C_VEL
LIN {X 0,Y 424.817,Z 439.689,A -85,B 0,C 180,E1 -9979.908,E2 -9979.908} C_VEL
LIN {X 0,Y 422.304,Z 433.453,A -85,B 0,C 180,E1 -9980.901,E2 -9980.901} C_VEL
LIN {X 0,Y 419.964,Z 426.735,A -85,B 0,C 180,E1 -9981.838,E2 -9981.838} C_VEL
LIN {X 0,Y 419.733,Z 422.251,A -85,B 0,C 180,E1 -9982.364,E2 -9982.364} C_VEL
LIN {X 0,Y 420.508,Z 411.521,A -85,B 0,C 180,E1 -9983.404,E2 -9983.404} C_VEL
LIN {X 0,Y 421.117,Z 400.5,A -85,B 0,C 180,E1 -9984.255,E2 -9984.255} C_VEL
LIN {X 0,Y 421.693,Z 388.317,A -85,B 0,C 180,E1 -9984.982,E2 -9984.982} C_VEL
LIN {X 0,Y 422.166,Z 375.779,A -85,B 0,C 180,E1 -9985.523,E2 -9985.523} C_VEL
LIN {X 0,Y 422.505,Z 362.291,A -85,B 0,C 180,E1 -9985.891,E2 -9985.891} C_VEL
LIN {X 0,Y 423.324,Z 279.3,A -85,B 0,C 180,E1 -9987.326,E2 -9987.326} C_VEL
LIN {X 0,Y 419.79,Z 259.064,A -85,B 0,C 180,E1 -9987.843,E2 -9987.843} C_VEL
LIN {X 0,Y 419.793,Z 257.485,A -85,B 0,C 180,E1 -9988.083,E2 -9988.083} C_VEL
LIN {X 0,Y 420.378,Z 246.665,A -85,B 0,C 180,E1 -9990.48,E2 -9990.48} C_VEL
LIN {X 0,Y 419.167,Z 238.515,A -85,B 0,C 180,E1 -9992.404,E2 -9992.404} C_VEL
LIN {X 0,Y 418.357,Z 234.935,A -85,B 0,C 180,E1 -9993.342,E2 -9993.342} C_VEL
